Universal Robots URScript: faichun_9jan_1t1.script

def faichun_9jan_1t1():
  set_tool_communication(True, 1000000, 2, 1, 1.5, 3.5)
  set_tool_output_mode(0)
  set_tool_digital_output_mode(0, 1)
  set_tool_digital_output_mode(1, 1)
  set_tool_voltage(24)
  step_count_e741a7f4_0b30_46a8_b996_4636aff9ce90 = 0.0
  thread Step_Counter_Thread_bd4b55fe_d110_495a_a627_b98bcdc962aa():
    while (True):
      step_count_e741a7f4_0b30_46a8_b996_4636aff9ce90 = step_count_e741a7f4_0b30_46a8_b996_4636aff9ce90 + 1.0
      sync()
    end
  end
  run Step_Counter_Thread_bd4b55fe_d110_495a_a627_b98bcdc962aa()
  set_gravity([0.0, 0.0, 9.82])
  set_tcp(p[0.0,0.0,0.0,0.0,0.0,0.0])
  set_standard_analog_input_domain(0, 1)
  set_standard_analog_input_domain(1, 1)
  set_tool_analog_input_domain(0, 1)
  set_tool_analog_input_domain(1, 1)
  set_analog_outputdomain(0, 0)
  set_analog_outputdomain(1, 0)
  set_input_actions_to_default()
  set_safety_mode_transition_hardness(1)
  set_target_payload(1.070000, [0.002000, 0.003000, 0.057000], [0.001723, 0.001723, 0.001723, 0.000000, 0.000000, 0.000000])
  global B1empty=False
  global A2Empty=0
  global A1Empty=0
  global B2Empty=False
  global pallet_step=0
  global bright_box=0
  global Pallet_1_cnt=2
  global dark_boxes=0
  global Point_1=p[0.6913645118948067,-0.12399382748223003,0.49223711947071,-1.2983729986843258,1.1259514972191385,-1.2203503861141718]
  # begin: URCap Installation Node
  #   Source: External Control, 1.0.5, FZI Research Center for Information Technology
  #   Type: External Control
  # end: URCap Installation Node
  # begin: URCap Installation Node
  #   Source: OnRobot, 6.2.0, OnRobot A/S
  #   Type: OnRobot Setup
  sleep(1)
  if (False):
  end
  ON_CONN_SHIFT_BOOL = 64
  ON_CONN_SHIFT_INT = 24
  ON_CONN_SHIFT_FLOAT = 24
  ON_CONN_REG_SUM_BOOL = 0
  ON_CONN_REG_SUM_INT = 1
  ON_CONN_REG_SUM_FLOAT = 0
  ON_TOOL_SHIFT_BOOL = 64
  ON_TOOL_SHIFT_INT = 25
  ON_TOOL_SHIFT_FLOAT = 24
  ON_TOOL_SHIFT_BOOL_ARR = [64, 64, 64]
  ON_TOOL_SHIFT_INT_ARR = [25, 25, 25]
  ON_TOOL_SHIFT_FLOAT_ARR = [24, 24, 24]
  ON_TOOL_REG_SUM_BOOL = 0
  ON_TOOL_REG_SUM_INT = 0
  ON_TOOL_REG_SUM_FLOAT = 0
  ON_REGISTERS_SPEEDL_FLOAT = 0
  ON_REG_USE_TOOL = False
  ON_DI_SINGLE = 0
  ON_DI_PRIMARY = 1
  ON_DI_SECONDARY = 2
  ON_DI_DUAL = 3
  on_robot_type = 10
  on_robot_cycle = 2.0
  on_conn_ip = "localhost"
  on_tool_ip = "localhost"
  on_device_socket_port = 51234
  on_conn_xmlrpc = rpc_factory("xmlrpc", "http://localhost:41414")
  on_tool_xmlrpc = rpc_factory("xmlrpc", "http://localhost:41414")
  on_RPC = rpc_factory("xmlrpc", "http://127.0.0.1:31416")
  ON_DEBUG_LOG = False
  on_isMetric = True
  on_toolConnector = True
  on_ioqc = False
  on_dual = False
  on_computebox = False
  on_devices = 0
  on_gripper = [False, False, False]
  on_custom_tcp_id = "none"
  on_custom_tcp_enabled = False
  speedlTime = 0.001
  on_ft = False
  #======    OnRobot Globals    ======#

  ON_MATH_PI=3.141593
  ON_ZEROPOSE=p[0.0,0.0,0.0,0.0,0.0,0.0]
  ON_ZEROFRAME=p[0.0,0.0,0.0,0.0,0.0,0.0]
  ON_ZERO3D=[0.0,0.0,0.0]
  ON_ZERO6D=[0.0,0.0,0.0,0.0,0.0,0.0]
  ON_ZERO8D=[0.0,0.0,0.0,0.0,0.0,0.0,0.0,0.0]
  ON_FALSE3D=[False,False,False]
  ON_FALSE6D=[False,False,False,False,False,False]
  ON_FALSE8D=[False,False,False,False,False,False,False,False]
  global on_return=0
  on_speedL=ON_ZERO6D
  on_speedBase=ON_ZERO6D
  on_speedVect=ON_ZERO6D
  on_speedExtra=ON_ZERO6D
  on_speedCB=ON_ZERO6D
  on_speedGecko=ON_ZERO6D
  on_RTDE_error=0
  on_RTDE_tool_error=0
  on_dataProcess_thrd=0
  ON_DEVICE_ID_MISSING=0
  ON_INIT_WATCHDOG_HZ=5
  ON_INIT_TIMEOUT=2000
  on_robot_TCP_offset=ON_ZEROFRAME
  on_tcp_offset_actual=ON_ZEROFRAME
  on_cog_actual=ON_ZEROFRAME
  on_mass_actual=0.0
  on_robot_mount=[0.0,0.0]

  #======    End of OnRobot Globals    ======#
  #======    OnRobot Interface Messages    ======#

  on_devices_primary_log="OnRobot Devices"
  on_devices_secondary_log="OnRobot Secondary Device"
  on_program_halted="<br>Program halted."
  on_device_error_title="OnRobot - Device error"
  on_install_error="OnRobot Setup is not correct.<br>Check the status in the OnRobot Setup page in the Installation Tab.<br>Program halted."
  on_device_missing="No device connected.<br>Program halted."
  cb_device_missing="No OnRobot Compute Box connected.<br>Program halted."
  ft_device_missing="No OnRobot FT sensor or license detected.<br>Program halted."
  hex_device_missing="No HEX sensor connected.<br>Program halted."
  rg2ft_device_missing="No RG2-FT gripper connected.<br>Program halted."
  rg_device_missing="No RG gripper connected.<br>Program halted."
  vg_device_missing="No VG gripper connected.<br>Program halted."
  gg_device_missing="No Gecko Gripper connected.<br>Program halted."
  sg_device_missing="No Soft Gripper connected.<br>Program halted."
  tfg_device_missing="No 3FG gripper connected.<br>Program halted."
  sdr_device_missing="No OnRobot Sander connected.<br>Program halted."
  twofg_device_missing="No 2FG gripper connected.<br>Program halted."
  vgp_device_missing="No VGP gripper connected.<br>Program halted."
  mg_device_missing="No Magnetic Gripper connected.<br>Program halted."
  fgp_device_missing="No 2FGP20 Gripper connected.<br>Program halted."
  eyes_device_missing="No OnRobot Eyes connected.<br>Program halted."
  on_xmlrpc_start_ip="Connecting to OnRobot XML-RPC Server:"
  on_java_comm_error_textmsg_title="OnRobot - Communication error:"
  on_java_comm_controlsocket_open_error="Socket 'javaSocket' opening was unsuccessful."
  on_java_comm_error_title="OnRobot - Communication error"
  on_java_comm_socket_open_error="Establishing connection with the URCap was timed out.<br>Check the status in the OnRobot Setup page in the Installation Tab.<br>Program halted."
  on_rtde_feed_error_textmsg_title="OnRobot - RTDE error:"
  on_rtde_feed_error="RTDE feed error. OnRobot device count mismatch.<br>Program halted."
  on_rtde_feed_tool_error="Tool RTDE feed error. OnRobot device count mismatch.<br>Program halted."
  on_rtde_feed_open_error_textmsg="Socket 'rtdeFeed' opening was unsuccessful."
  on_rtde_feed_error_title="OnRobot - RTDE error"
  on_rtde_feed_count_error="Invalid RTDE offset setup detected. Please check RTDE Offsets at the OnRobot Setup page in the Installation Tab.<br>Program halted."
  on_rtde_feed_open_error="Establishing connection with the devices was timed out.<br>Ensure that the OnRobot devices are operational, and check the status in the OnRobot Setup page in the Installation Tab."

  #======    End of OnRobot Interface Messages    ======#
  #======    OnRobot Interface    ======#

  on_portopened_javaSocket=False
  on_rtde_feed_opened=False
  on_dataProcess_running=False
  def on_missing():
  popup(on_device_missing,title=on_device_error_title,error=True,blocking=False)
  halt
  end
  def cb_missing():
  popup(cb_device_missing,title=on_device_error_title,error=True,blocking=False)
  halt
  end
  def ft_missing():
  popup(ft_device_missing,title=on_device_error_title,error=True,blocking=False)
  halt
  end
  def hex_missing():
  popup(hex_device_missing,title=on_device_error_title,error=True,blocking=False)
  halt
  end
  def rg2ft_missing():
  popup(rg2ft_device_missing,title=on_device_error_title,error=True,blocking=False)
  halt
  end
  def rg_missing():
  popup(rg_device_missing,title=on_device_error_title,error=True,blocking=False)
  halt
  end
  def vg_missing():
  popup(vg_device_missing,title=on_device_error_title,error=True,blocking=False)
  halt
  end
  def gg_missing():
  popup(gg_device_missing,title=on_device_error_title,error=True,blocking=False)
  halt
  end
  def sg_missing():
  popup(sg_device_missing,title=on_device_error_title,error=True,blocking=False)
  halt
  end
  def tfg_missing():
  popup(tfg_device_missing,title=on_device_error_title,error=True,blocking=False)
  halt
  end
  def sdr_missing():
  popup(sdr_device_missing,title=on_device_error_title,error=True,blocking=False)
  halt
  end
  def twofg_missing():
  popup(twofg_device_missing,title=on_device_error_title,error=True,blocking=False)
  halt
  end
  def vgp_missing():
  popup(vgp_device_missing,title=on_device_error_title,error=True,blocking=False)
  halt
  end
  def mg_missing():
  popup(mg_device_missing,title=on_device_error_title,error=True,blocking=False)
  halt
  end
  def fgp_missing():
  popup(fgp_device_missing,title=on_device_error_title,error=True,blocking=False)
  halt
  end
  def eyes_missing():
  popup(eyes_device_missing,title=on_device_error_title,error=True,blocking=False)
  halt
  end
  def on_portclose_javaSocket():
  socket_close("javaSocket")
  on_portopened_javaSocket=False
  end
  def on_portopen_javaSocket():
  on_portclose_javaSocket()
  on_portopened_javaSocket=socket_open("127.0.0.1",44005,"javaSocket")
  if not on_portopened_javaSocket:
  textmsg(on_java_comm_error_textmsg_title,on_java_comm_controlsocket_open_error)
  popup(on_java_comm_socket_open_error,title=on_java_comm_error_title,error=True,blocking=False)
  halt
  end
  end
  on_conn_rtde_feed_name="rtdeFeedConn"
  on_tool_rtde_feed_name="rtdeFeedTool"
  def on_rtde_feed_close(rtdeFeedName):
  socket_close(rtdeFeedName)
  on_rtde_feed_opened=False
  end
  def on_rtde_feed_open(deviceIP,rtdeFeedName,regStart,regSum,regSpeedl):
  on_rtde_feed_close(rtdeFeedName)
  if((regStart[0]+regSum[0])>128)or((regStart[1]+regSum[1])>48)or((regStart[2]+regSum[2])>48):
  popup(on_rtde_feed_count_error,title=on_rtde_feed_error_title,error=True,blocking=False)
  textmsg(str_cat("RegStart: ",regStart),str_cat("  -  RegSum: ",regSum))
  halt
  end
  on_rtde_feed_opened=socket_open(deviceIP,on_device_socket_port,rtdeFeedName)
  if not on_rtde_feed_opened:
  on_rtde_feed_opened=socket_open(deviceIP,on_device_socket_port,rtdeFeedName)
  end
  if not on_rtde_feed_opened:
  textmsg(on_rtde_feed_error_textmsg_title,on_rtde_feed_open_error_textmsg)
  popup(on_rtde_feed_open_error,title=on_rtde_feed_error_title,error=True,blocking=False)
  halt
  end
  socket_send_int(regStart[0],rtdeFeedName)
  socket_send_int(regSum[0],rtdeFeedName)
  socket_send_int(regStart[1],rtdeFeedName)
  socket_send_int(regSum[1],rtdeFeedName)
  socket_send_int(regStart[2],rtdeFeedName)
  socket_send_int(regSum[2],rtdeFeedName)
  socket_send_int(regSpeedl,rtdeFeedName)
  socket_send_int(on_devices,rtdeFeedName)
  end
  def on_dataRead():
  enter_critical
  on_RTDE_error=read_input_integer_register(ON_CONN_SHIFT_INT)
  if(ON_REG_USE_TOOL):
  on_RTDE_tool_error=read_input_integer_register(ON_TOOL_SHIFT_INT_ARR[0])
  end
  exit_critical
  end
  def on_set_rtde_watchdog(updateHz=ON_INIT_WATCHDOG_HZ):
  local effect="stop"
  if(updateHz<1):
  effect="ignore"
  end
  watchdog_conn_reg_str=str_cat("input_int_register_",ON_CONN_SHIFT_INT)
  rtde_set_watchdog(watchdog_conn_reg_str,updateHz,effect)
  if(ON_REG_USE_TOOL):
  watchdog_tool_reg_str=str_cat("input_int_register_",ON_TOOL_SHIFT_INT_ARR[0])
  rtde_set_watchdog(watchdog_tool_reg_str,updateHz,effect)
  end
  if ON_DEBUG_LOG:
  local update_str=str_cat(" "+effect+" watchdog set to [Hz]: ",updateHz)
  textmsg(watchdog_conn_reg_str,update_str)
  if(ON_REG_USE_TOOL):
  local update_str=str_cat(" "+effect+" watchdog set to [Hz]: ",updateHz)
  textmsg(watchdog_tool_reg_str,update_str)
  end
  end
  end
  def on_speedCB_get():
  return[on_speedCB[0],on_speedCB[1],on_speedCB[2],on_speedCB[3],on_speedCB[4],on_speedCB[5]]
  end
  def on_speedGecko_get():
  local speedExtra=ON_ZERO6D
  if on_speedl_for_gecko:
  speedExtra=[on_speedGecko[0],on_speedGecko[1],on_speedGecko[2],on_speedGecko[3],on_speedGecko[4],on_speedGecko[5]]
  end
  return speedExtra
  end
  def on_speedGecko_set(speedGecko):
  on_speedGecko=[speedGecko[0],speedGecko[1],speedGecko[2],speedGecko[3],speedGecko[4],speedGecko[5]]
  end
  thread on_dataProcess_thread():
  if ON_DEBUG_LOG:
  textmsg("Starting on_dataRead thread")
  end
  local error=False
  on_dataProcess_running=True
  sync()
  while on_dataProcess_running:
  sync()
  on_dataRead()
  error=on_error((on_RTDE_error<0),on_rtde_feed_error,on_rtde_feed_error_title,error)
  error=on_error((ON_REG_USE_TOOL and(on_RTDE_tool_error<0)),on_rtde_feed_tool_error,on_rtde_feed_error_title,error)
  on_dataProcess_running=not error
  end
  if error:
  halt
  end
  if ON_DEBUG_LOG:
  textmsg("Stopping on_dataRead thread")
  end
  end
  thread on_set_watchdog_thread():
  sleep(2)
  on_set_rtde_watchdog(updateHz=ON_INIT_WATCHDOG_HZ)
  sleep(1/ON_INIT_WATCHDOG_HZ)
  on_dataProcess_running=False
  kill on_dataProcess_thrd
  end

  #======    End of OnRobot Interface    ======#
  #======    OnRobot QC Setup Tool Connector    ======#

  def tc_setup_tool():
  if ON_DEBUG_LOG:
  textmsg("QC Setup Tool Connector start...")
  end
  set_tool_voltage(24)

  set_tool_communication(True,1000000,2,1,1.5,3.5)

  if ON_DEBUG_LOG:
  textmsg("QC Setup Tool Connector end.")
  end
  end

  #======    End of OnRobot QC Setup Tool Connector    ======#
  #======    OnRobot TCP Messages    ======#

  on_tcp_log_msg_default="OnRobot: Robot TCP Offset set to:"
  on_tcp_log_msg_primary="OnRobot: Robot TCP Offset set to Primary:"
  on_tcp_log_msg_secondary="OnRobot: Robot TCP Offset set to Secondary:"

  #======    End of OnRobot TCP Messages    ======#
  #======    OnRobot TCP    ======#

  on_tcp_offset_actual=ON_ZEROFRAME
  on_tcp_offset_primary=ON_ZEROFRAME
  on_tcp_static_primary=ON_ZEROFRAME
  on_tcp_dynamic_primary=ON_ZEROFRAME
  on_tcp_adapters=ON_ZEROFRAME
  on_tcp_qc_primary=ON_ZEROFRAME
  on_tcp_base_primary=ON_ZEROFRAME
  on_tcp_gripper_static_primary=ON_ZEROFRAME
  on_tcp_workpiece_primary=ON_ZEROFRAME
  on_tcp_gripper_dynamic_primary=ON_ZEROFRAME
  on_tcp_gripper_primary=ON_ZEROFRAME
  on_tcp_offset_secondary=ON_ZEROFRAME
  on_tcp_static_secondary=ON_ZEROFRAME
  on_tcp_dynamic_secondary=ON_ZEROFRAME
  on_tcp_qc_secondary=ON_ZEROFRAME
  on_tcp_base_secondary=ON_ZEROFRAME
  on_tcp_gripper_static_secondary=ON_ZEROFRAME
  on_tcp_workpiece_secondary=ON_ZEROFRAME
  on_tcp_gripper_dynamic_secondary=ON_ZEROFRAME
  on_tcp_gripper_secondary=ON_ZEROFRAME
  on_tcp_custom_preset_assigned=False
  on_tcp_custom_preset=ON_ZEROFRAME
  def on_tcp_init_adapters():
  if ON_DEBUG_LOG:
  textmsg("TCP Init Adapters start..")
  end
  enter_critical
  on_tcp_adapters=ON_ZEROFRAME
  local adapterCount=length(on_tcp_adapters_array)
  local i=0
  while(i<adapterCount):
  on_tcp_adapters=pose_trans(on_tcp_adapters,on_tcp_adapters_array[i])
  i=i+1
  end
  exit_critical
  if ON_DEBUG_LOG:
  textmsg("TCP Init Adapters end.")
  end
  end
  def on_tcp_update_primary():
  if ON_DEBUG_LOG:
  textmsg("TCP Update Primary start..")
  end
  on_tcp_gripper_dynamic_primary=p[0.0, 0.0, 0.0, 0.0, 0.0, 0.0]
  enter_critical
  on_tcp_dynamic_primary=pose_trans(on_tcp_static_primary,on_tcp_gripper_dynamic_primary)
  on_tcp_offset_primary=pose_trans(on_tcp_dynamic_primary,on_tcp_workpiece_primary)
  exit_critical
  if ON_DEBUG_LOG:
  textmsg("TCP Update Primary end.")
  end
  end
  def on_tcp_init_primary():
  if ON_DEBUG_LOG:
  textmsg("TCP Init Primary start..")
  end
  enter_critical
  on_tcp_base_primary=pose_trans(on_tcp_adapters,on_tcp_qc_primary)
  on_tcp_static_primary=pose_trans(on_tcp_base_primary,on_tcp_gripper_static_primary)
  exit_critical
  on_tcp_update_primary()
  if ON_DEBUG_LOG:
  textmsg("TCP Init Primary end.")
  end
  end
  def on_tcp_offset_set(TCP_offset):
  if ON_DEBUG_LOG:
  textmsg("TCP Offset set started!")
  end
  on_tcp_offset_send(TCP_offset)
  if(on_follow_tcp):
  set_tcp(TCP_offset)
  end
  on_robot_TCP_offset=TCP_offset
  if ON_DEBUG_LOG:
  textmsg("TCP Offset set to: ",on_robot_TCP_offset)
  end
  end
  def on_tcp_offset_forced_set_actual(isPrimary=True):
  if(not on_follow_tcp):

  local tcp_log_msg=on_tcp_log_msg_default

  textmsg(tcp_log_msg,on_tcp_offset_actual)
  set_tcp(on_tcp_offset_actual)
  end
  end
  def on_tcp_update(isPrimary=True):
  on_tcp_update_primary()

  on_tcp_set_actual_to(isPrimary)
  end
  def on_tcp_set_actual_to(isPrimary=True):

  on_tcp_offset_actual=on_tcp_offset_primary
  if(on_follow_tcp):
  textmsg(on_tcp_log_msg_default,on_tcp_offset_actual)
  end

  on_tcp_active_is_primary=isPrimary
  on_tcp_offset_set(on_tcp_offset_actual)
  end
  def on_tcp_update_workpiece_primary(workpiece_offset):
  if ON_DEBUG_LOG:
  textmsg("TCP Update Tool Primary start..")
  end
  on_tcp_workpiece_primary=workpiece_offset
  on_tcp_update_primary()
  if ON_DEBUG_LOG:
  textmsg("TCP Update Tool Primary end.")
  end
  end
  def on_tcp_workpiece_rpy_get(xyz=[0.0,0.0,0.0],rpy=[0.0,0.0,0.0]):
  local rotvec=rpy2rotvec(rpy)
  local workpiece_offset=p[xyz[0],xyz[1],xyz[2],rotvec[0],rotvec[1],rotvec[2]]
  return workpiece_offset
  end

  def on_tcp_update_workpiece(workpiece_offset,tool_index=0):
  if ON_DEBUG_LOG:
  textmsg("TCP Update Tool start..")
  end
  if(tool_index!=ON_DI_SECONDARY):
  on_tcp_update_workpiece_primary(workpiece_offset)
  local isPrimary=True

  end
  on_tcp_set_actual_to(isPrimary)
  if ON_DEBUG_LOG:
  textmsg("TCP Update Tool end.")
  end
  end
  def on_get_tcp_for(tool_index):
  if tool_index==ON_DI_SECONDARY:
  local actual_tcp=on_tcp_static_secondary
  else:
  local actual_tcp=on_tcp_static_primary
  end
  return actual_tcp
  end
  def on_tcp_custom_unused():
  return ON_ZEROFRAME
  end
  def on_tcp_update_custom():
  if ON_DEBUG_LOG:
  textmsg("TCP Update Custom start..")
  end
  if(on_custom_tcp_enabled):
  on_tcp_custom_unused()
  on_tcp_custom_unused()
  on_tcp_custom_unused()
  on_tcp_custom_unused()

  end
  if ON_DEBUG_LOG:
  textmsg("TCP Update Custom end.")
  end
  end

  #======    End of OnRobot TCP    ======#
  #======    OnRobot Payload Messages    ======#

  on_mass_log_msg="OnRobot: Robot Payload Mass set to:"
  on_cog_log_msg="OnRobot: Robot Payload Center of Gravity set to:"

  #======    End of OnRobot Payload Messages    ======#
  #======    OnRobot Payload    ======#

  on_cog_actual=ON_ZEROFRAME
  on_mass_actual=0.0
  on_cog_primary=ON_ZEROFRAME
  on_cog_L1L2_primary=ON_ZEROFRAME
  on_mass_primary=0.0
  on_mass_L1L2_primary=0.0
  on_cog_adapters=ON_ZEROFRAME
  on_cog_qc_primary=ON_ZEROFRAME
  on_cog_base_primary=ON_ZEROFRAME
  on_cog_gripper_primary=ON_ZEROFRAME
  on_cog_workpiece_primary=ON_ZEROFRAME
  on_mass_adapters=0.0
  on_mass_qc_primary=0.0
  on_mass_base_primary=0.0
  on_mass_gripper_primary=0.0
  on_mass_workpiece_primary=0.0
  on_cog_secondary=ON_ZEROFRAME
  on_mass_secondary=0.0
  on_cog_gripper_secondary=ON_ZEROFRAME
  on_mass_gripper_secondary=0.0
  on_cog_workpiece_secondary=ON_ZEROFRAME
  on_mass_workpiece_secondary=0.0
  ON_LB2KG001=0.45359237/100
  def on_payload_init_adapters():
  if ON_DEBUG_LOG:
  textmsg("TCP Init Adapters start..")
  end
  enter_critical
  on_cog_adapters=ON_ZEROFRAME
  on_mass_adapters=0.0
  local massLAL0Ratio=0
  local adapterAbsCOG=ON_ZEROFRAME
  local tcp_adapter_offset=ON_ZEROFRAME
  local adapterCount=length(on_tcp_adapters_array)
  local i=0
  while(i<adapterCount):
  on_mass_adapters=on_mass_adapters+on_mass_adapters_array[i]
  if(on_mass_adapters<=0):
  massLAL0Ratio=0
  else:
  massLAL0Ratio=on_mass_adapters_array[i]/on_mass_adapters
  end
  adapterAbsCOG=pose_trans(tcp_adapter_offset,on_tcp_adapters_array[i])
  adapterAbsCOG=p[adapterAbsCOG[0],adapterAbsCOG[1],adapterAbsCOG[2],0.0,0.0,0.0]
  on_cog_adapters=interpolate_pose(on_cog_adapters,adapterAbsCOG,massLAL0Ratio)
  on_cog_adapters=p[on_cog_adapters[0],on_cog_adapters[1],on_cog_adapters[2],0.0,0.0,0.0]
  tcp_adapter_offset=pose_trans(tcp_adapter_offset,on_tcp_adapters_array[i])
  i=i+1
  sync()
  end
  exit_critical
  if ON_DEBUG_LOG:
  textmsg("TCP Init Adapters end.")
  end
  end
  def on_payload_update_primary():
  if ON_DEBUG_LOG:
  textmsg("Payload Update Primary start..")
  end
  enter_critical
  on_mass_primary=on_mass_L1L2_primary+on_mass_workpiece_primary
  local massL1L2L3Ratio=on_mass_workpiece_primary/on_mass_primary
  local workpieceAbsCOG=pose_trans(on_tcp_dynamic_primary,on_cog_workpiece_primary)
  workpieceAbsCOG=p[workpieceAbsCOG[0],workpieceAbsCOG[1],workpieceAbsCOG[2],0.0,0.0,0.0]
  on_cog_primary=interpolate_pose(on_cog_L1L2_primary,workpieceAbsCOG,massL1L2L3Ratio)
  on_cog_primary=p[on_cog_primary[0],on_cog_primary[1],on_cog_primary[2],0.0,0.0,0.0]
  exit_critical
  if ON_DEBUG_LOG:
  textmsg("Payload Update Primary end.")
  end
  end
  def on_payload_init_primary():
  if ON_DEBUG_LOG:
  textmsg("Payload Init Primary start..")
  end
  enter_critical
  on_mass_base_primary=on_mass_adapters+on_mass_qc_primary
  local massL0L1Ratio=on_mass_qc_primary/on_mass_base_primary
  on_mass_L1L2_primary=on_mass_base_primary+on_mass_gripper_primary
  local massL1L2Ratio=on_mass_gripper_primary/on_mass_L1L2_primary
  local qcAbsCOG=pose_trans(on_tcp_adapters,on_cog_qc_primary)
  qcAbsCOG=p[qcAbsCOG[0],qcAbsCOG[1],qcAbsCOG[2],0.0,0.0,0.0]
  on_cog_base_primary=interpolate_pose(on_cog_adapters,qcAbsCOG,massL0L1Ratio)
  on_cog_base_primary=p[on_cog_base_primary[0],on_cog_base_primary[1],on_cog_base_primary[2],0.0,0.0,0.0]
  local gripperAbsCOG=pose_trans(on_tcp_base_primary,on_cog_gripper_primary)
  gripperAbsCOG=p[gripperAbsCOG[0],gripperAbsCOG[1],gripperAbsCOG[2],0.0,0.0,0.0]
  on_cog_L1L2_primary=interpolate_pose(on_cog_base_primary,gripperAbsCOG,massL1L2Ratio)
  on_cog_L1L2_primary=p[on_cog_L1L2_primary[0],on_cog_L1L2_primary[1],on_cog_L1L2_primary[2],0.0,0.0,0.0]
  exit_critical
  on_payload_update_primary()
  if ON_DEBUG_LOG:
  textmsg("Payload Init Primary end.")
  end
  end
  def on_payload_update():
  on_payload_update_primary()

  on_mass_actual =on_mass_primary
  on_cog_actual=on_cog_primary

  on_payload_set_actual()
  end
  def on_payload_set_actual():

  on_mass_actual =on_mass_primary
  on_cog_actual=on_cog_primary

  local CoG=[on_cog_actual[0],on_cog_actual[1],on_cog_actual[2]]
  on_payload_set(on_mass_actual,CoG)
  end
  def on_payload_update_workpiece_primary(workpiece_mass=0,workpiece_cog=[0.0,0.0,0.0]):
  if ON_DEBUG_LOG:
  textmsg("Payload Update Workpiece Primary start..")
  end
  on_cog_workpiece_primary=p[workpiece_cog[0],workpiece_cog[1],workpiece_cog[2],0.0,0.0,0.0]
  on_mass_workpiece_primary=workpiece_mass
  on_payload_update_primary()
  if ON_DEBUG_LOG:
  textmsg("Payload Update Workpiece Primary end.")
  end
  end
  def on_payload_set(mass,CoG):
  if ON_DEBUG_LOG:
  textmsg("Payload set started!")
  end
  local center_of_gravity=[CoG[0],CoG[1],CoG[2]]
  on_payload_send(center_of_gravity,mass)
  if(on_isMetric):
  local roundedMass=floor(mass*100+0.5)/100
  else:
  local roundedMass=floor(mass/ON_LB2KG001+0.5)*ON_LB2KG001
  end
  set_payload(roundedMass,center_of_gravity)
  on_mass_actual=roundedMass
  on_cog_actual=p[CoG[0],CoG[1],CoG[2],0.0,0.0,0.0]
  if ON_DEBUG_LOG:
  textmsg("Payload mass, CoG set to: ",str_cat(str_cat(mass,", "),CoG))
  end
  end

  def on_payload_update_secondary():
  end
  def on_payload_init_secondary():
  end

  def on_payload_update_workpiece(workpiece_mass,workpiece_cog=[0.0,0.0,0.0],tool_index=0):
  if ON_DEBUG_LOG:
  textmsg("Payload Update Workpiece start..")
  end
  if(tool_index!=ON_DI_SECONDARY):
  on_cog_workpiece_primary=p[workpiece_cog[0],workpiece_cog[1],workpiece_cog[2],0.0,0.0,0.0]
  on_mass_workpiece_primary=workpiece_mass
  else:
  on_cog_workpiece_secondary=p[workpiece_cog[0],workpiece_cog[1],workpiece_cog[2],0.0,0.0,0.0]
  on_mass_workpiece_secondary=workpiece_mass
  end
  on_payload_update()
  if ON_DEBUG_LOG:
  textmsg("Payload Update Workpiece end.")
  end
  end
  def on_payload_get_cog2tcp_workpiece(tool_index=0):
  if(tool_index!=ON_DI_SECONDARY):
  local cog_tool=[on_tcp_workpiece_primary[0],on_tcp_workpiece_primary[1],on_tcp_workpiece_primary[2]]
  else:
  local cog_tool=[on_tcp_workpiece_secondary[0],on_tcp_workpiece_secondary[1],on_tcp_workpiece_secondary[2]]
  end
  return cog_tool
  end

  #======    End of OnRobot Payload    ======#
  #======    OnRobot QC TCP    ======#

  onrobotmini=0

  def on_tcp_offset_send(TCP_offset):
  on_robot_TCP_offset=TCP_offset
  end
  def on_payload_send(CoG,mass):
  on_robot_payload_cog=CoG
  on_robot_payload_mass=mass
  end


  #======    End of OnRobot QC TCP    ======#
  #======    OnRobot  Speedl    ======#

  on_speedl_thread_handler=0
  on_speedl_is_enabled=False
  on_speedl_is_running=False
  on_speedl_acc=0.0
  ft_speedl_hg_caranteen_reached=False
  ft_speedl_hg_caranteen_safemode=False
  on_speedl_for_ftcontrol=False
  on_speedl_for_move=False
  on_speedl_for_handguide=False
  on_speedl_for_insertpart=False
  on_speedl_for_depthcompensation=False
  on_speedl_for_center=False
  on_speedl_for_gecko=False
  on_speedl_acc=10000.0
  on_speedl_acc_to_zero=3.0
  ON_SPEEDL_FTCONTROL=1
  ON_SPEEDL_HANDGUIDE=2
  ON_SPEEDL_TRAJECTORY=3
  ON_SPEEDL_MOVE=ON_SPEEDL_TRAJECTORY
  ON_SPEEDL_INSERTPART=4
  ON_SPEEDL_DEPTHCOMP=5
  ON_SPEEDL_CENTER=6
  ON_SPEEDL_GECKO=7
  def on_wait_ms(time_ms):
  local sync_time=ceil(norm(time_ms/2.0))
  while(sync_time>0):
  sync_time=sync_time-1
  sync()
  end
  end
  def on_error(status_flag,message,title,stop_var=False):
  if(status_flag):
  popup(message,title=title,error=True,blocking=False)
  stop_var=True
  end
  return stop_var
  end
  def on_warning(status_flag,message,title,isPopupNeeded=False,is_shown=False):
  if(status_flag):
  if(not is_shown):
  if(isPopupNeeded):
  popup(message,title=title,warning=True,blocking=False)
  else:
  textmsg(title+": ",message)
  end
  is_shown=True
  end
  else:
  is_shown=False
  end
  return is_shown
  end
  def on_speedl_add_extra(speedBase,speedExtra):
  speedSum=ON_ZERO6D
  speedBaseP=p[speedBase[0],speedBase[1],speedBase[2],speedBase[3],speedBase[4],speedBase[5]]
  speedExtraP=p[speedExtra[0],speedExtra[1],speedExtra[2],speedExtra[3],speedExtra[4],speedExtra[5]]
  speedSumP=pose_add(speedExtraP,speedBaseP)
  speedSum=[speedSumP[0],speedSumP[1],speedSumP[2],speedSumP[3],speedSumP[4],speedSumP[5]]
  return speedSum
  end

  thread on_speedl_thread():
  if ON_DEBUG_LOG:
  textmsg("Speedl thread started..")
  end
  enter_critical
  on_speedl_is_running=True
  on_speedl_is_enabled=True
  exit_critical
  on_speedL=ON_ZERO6D
  on_speedL_last=ON_ZERO6D

  while on_speedl_is_running:
  on_speedBase=on_speedCB_get()
  on_speedL=on_speedBase


  if on_speedl_is_enabled:
  if(on_speedL==ON_ZERO6D):
  on_speedL=[on_speedL_last[0]/100,on_speedL_last[1]/100,on_speedL_last[2]/100,on_speedL_last[3]/100,on_speedL_last[4]/100,on_speedL_last[5]/100]
  end
  speedl(on_speedL,a=on_speedl_acc,t=speedlTime)
  else:
  speedl(ON_ZERO6D,a=on_speedl_acc_to_zero,t=speedlTime)
  end
  on_speedL_last=on_speedL
  end

  on_speedL=ON_ZERO6D
  if ON_DEBUG_LOG:
  textmsg("Speedl thread ended.")
  end
  end
  def on_speedl_integer_get():
  local speedl_integer=binary_list_to_integer([on_speedl_for_ftcontrol,on_speedl_for_handguide,on_speedl_for_move,on_speedl_for_insertpart,on_speedl_for_depthcompensation,on_speedl_for_center,on_speedl_for_gecko])
  return speedl_integer
  end
  def on_speedl_start_for(speedl_id):
  if(speedl_id==ON_SPEEDL_FTCONTROL):
  on_speedl_for_ftcontrol=True
  elif(speedl_id==ON_SPEEDL_HANDGUIDE):
  on_speedl_for_handguide=True
  elif(speedl_id==ON_SPEEDL_TRAJECTORY):
  on_speedl_for_move=True
  elif(speedl_id==ON_SPEEDL_INSERTPART):
  on_speedl_for_insertpart=True
  elif(speedl_id==ON_SPEEDL_DEPTHCOMP):
  on_speedl_for_depthcompensation=True
  elif(speedl_id==ON_SPEEDL_CENTER):
  on_speedl_for_center=True
  elif(speedl_id==ON_SPEEDL_GECKO):
  on_speedl_for_gecko=True
  else:
  textmsg("Unknown Start speedl ID received: ",speedl_id)
  end
  local speedl_integer=on_speedl_integer_get()
  if not(speedl_integer==0):
  if not on_speedl_is_running:
  on_speedl_thread_handler=run on_speedl_thread()
  end
  end
  return on_speedl_is_running
  end
  def on_speedl_stop_for(speedl_id,brake=10,brakeRot=10):
  if(speedl_id==ON_SPEEDL_FTCONTROL):
  on_speedl_for_ftcontrol=False
  elif(speedl_id==ON_SPEEDL_HANDGUIDE):
  on_speedl_for_handguide=False
  elif(speedl_id==ON_SPEEDL_TRAJECTORY):
  on_speedl_for_move=False
  elif(speedl_id==ON_SPEEDL_INSERTPART):
  on_speedl_for_insertpart=False
  elif(speedl_id==ON_SPEEDL_DEPTHCOMP):
  on_speedl_for_depthcompensation=False
  elif(speedl_id==ON_SPEEDL_CENTER):
  on_speedl_for_center=False
  elif(speedl_id==ON_SPEEDL_GECKO):
  on_speedl_for_gecko=False
  on_speedGecko_set(ON_ZERO6D)
  else:
  textmsg("Unknown Stop speedl ID received: ",speedl_id)
  end
  local speedl_integer=on_speedl_integer_get()
  if(speedl_integer==0):
  if(on_speedl_is_running):
  kill on_speedl_thread_handler
  enter_critical
  on_speedl_is_running=False
  exit_critical

  end
  if ON_DEBUG_LOG:
  textmsg("Speedl thread stopped")
  end
  stopl(brake,brakeRot)
  end
  return on_speedl_is_running
  end
  def on_speedl_pause():
  on_speedl_is_enabled=False
  return on_speedl_integer_get()
  end
  def on_speedl_resume():
  on_speedl_is_enabled=True
  return on_speedl_integer_get()
  end

  #======    End of OnRobot  Speedl    ======#
  textmsg(on_devices_primary_log, ": Quick Changer + QC Tool Side + [0.0, 0.0, 0.0, 0.0, 0.0, 0.0]")
  on_follow_tcp = False
  on_tcp_active_is_primary = True
  on_tcp_adapters_array = []
  on_cog_adapters_array = []
  on_mass_adapters_array = []
  on_tcp_qc_primary = p[0.0, 0.0, 0.0136, 0.0, 0.0, 0.0]
  on_cog_qc_primary = p[0.0, 0.0, 0.004, 0.0, 0.0, 0.0]
  on_mass_qc_primary = 0.06
  on_tcp_gripper_static_primary = p[0.0, 0.0, 0.017, 0.0, 0.0, 0.0]
  on_cog_gripper_primary = p[0.0, 0.0, 0.002, 0.0, 0.0, 0.0]
  on_mass_gripper_primary = 0.14
  on_tcp_workpiece_primary = p[0.0, 0.0, 0.0, 0.0, 0.0, 0.0]
  on_cog_workpiece_primary = p[0.0, 0.0, 0.0, 0.0, 0.0, 0.0]
  on_mass_workpiece_primary = 0.0
  #======    OnRobot Run    ======#

  on_portopen_javaSocket()
  sync()
  textmsg(on_xmlrpc_start_ip,on_conn_ip)
  if(ON_REG_USE_TOOL):
  on_regStart_conn=[ON_CONN_SHIFT_BOOL,ON_CONN_SHIFT_INT,ON_CONN_SHIFT_FLOAT]
  on_regSum_conn=[ON_CONN_REG_SUM_BOOL,ON_CONN_REG_SUM_INT,ON_CONN_REG_SUM_FLOAT]
  on_rtde_feed_open(on_conn_ip,on_conn_rtde_feed_name,on_regStart_conn,on_regSum_conn,ON_REGISTERS_SPEEDL_FLOAT)
  sync()
  textmsg(on_xmlrpc_start_ip,on_tool_ip)
  on_regStart_tool=[ON_TOOL_SHIFT_BOOL,ON_TOOL_SHIFT_INT,ON_TOOL_SHIFT_FLOAT]
  on_regSum_tool=[ON_TOOL_REG_SUM_BOOL,ON_TOOL_REG_SUM_INT,ON_TOOL_REG_SUM_FLOAT]
  on_rtde_feed_open(on_tool_ip,on_tool_rtde_feed_name,on_regStart_tool,on_regSum_tool,0)
  sync()
  else:
  on_regStart_conn=[ON_CONN_SHIFT_BOOL,ON_CONN_SHIFT_INT,ON_CONN_SHIFT_FLOAT]
  on_regSum_conn=[ON_CONN_REG_SUM_BOOL,ON_CONN_REG_SUM_INT,ON_CONN_REG_SUM_FLOAT]
  on_rtde_feed_open(on_conn_ip,on_conn_rtde_feed_name,on_regStart_conn,on_regSum_conn,ON_REGISTERS_SPEEDL_FLOAT)
  sync()
  end
  on_set_rtde_watchdog(updateHz=0.2)
  sync()
  on_dataProcess_thrd=run on_dataProcess_thread()
  sync()
  on_tcp_init_adapters()
  on_payload_init_adapters()
  on_tcp_init_primary()
  on_payload_init_primary()

  on_tcp_update_custom()
  on_tcp_set_actual_to(on_tcp_active_is_primary)
  if(on_follow_tcp):
  on_payload_set_actual()
  end
  on_watchdog_thrd=run on_set_watchdog_thread()
  sync()
  def done_waiting_for_init(device_name,product_code,tool_index=0):
  textmsg(str_cat(device_name,str_cat(str_cat("[",tool_index),"]: ")),product_code)
  end

  #======    End of OnRobot Run    ======#
  #======    OnRobot QC Start    ======#

  if(on_toolConnector):
  tc_setup_tool()
  end
  sync()

  #======    End of OnRobot QC Start    ======#
  # end: URCap Installation Node
  $ 1 "Robot Program"
  $ 2 "Script: FaiChun_9 Jan_11_2_t1.script"
  def Machining1():
    # Default parameters:
    global speed_ms = 0.05
    global speed_rads = 0.75
    global accel_mss = 3
    global accel_radss = 1.2
    global blend_radius_m = 0.0003

    # Add subprograms here
    # Start of main program
    # Program generated by RoboDK v5.6.8 for UR10e on 17/01/2025 15:24:14
    # Using nominal kinematics.
    blend_radius_m = 0.0003
    speed_ms = 0.05
    # set_reference(p[0.340000, -0.240000, 0.001500, 0.000000, 0.000000, 0.000000])
    set_tcp(p[0.000000, 0.000000, 0.252000, 0.000000, 0.000000, 0.000000])
    # Show Tool
    movej([0.140721, -1.398447, -2.445688, -0.868253, 1.570796, 1.711517],accel_radss,speed_rads,0,blend_radius_m)
    movel([0.140721, -1.451124, -2.475554, -0.785711, 1.570796, 1.711517],accel_mss,speed_ms,0,blend_radius_m)
    #SetTool1
    #M_RunCode6
    #SetRPM60000
    speed_ms = 0.05
    #M_RunCode3
    movel([0.140721, -1.474076, -2.486639, -0.751674, 1.570796, 1.711517],accel_mss,speed_ms,0,blend_radius_m)
    speed_ms = 0.003
    movel([0.140721, -1.480003, -2.489338, -0.743048, 1.570796, 1.711517],accel_mss,speed_ms,0,blend_radius_m)
    speed_ms = 0.02
    movel([-0.135603, -1.563113, -2.412732, -0.736544, 1.570796, 1.435194],accel_mss,speed_ms,0,blend_radius_m)
    movel([-0.182919, -1.334068, -2.598334, -0.779987, 1.570796, 1.387878],accel_mss,speed_ms,0,blend_radius_m)
    movel([0.198662, -1.168946, -2.687374, -0.856069, 1.570796, 1.769459],accel_mss,speed_ms,0,blend_radius_m)
    movel([0.140721, -1.480003, -2.489338, -0.743048, 1.570796, 1.711517],accel_mss,speed_ms,0,blend_radius_m)
    speed_ms = 0.003
    movel([0.140721, -1.474076, -2.486639, -0.751674, 1.570796, 1.711517],accel_mss,speed_ms,0,blend_radius_m)
    speed_ms = 0.05
    movel([0.140721, -1.451124, -2.475554, -0.785711, 1.570796, 1.711517],accel_mss,speed_ms,0,blend_radius_m)
    #M_RunCode9
    movel([0.136570, -1.444454, -2.480985, -0.786951, 1.570796, 1.707367],accel_mss,speed_ms,0,blend_radius_m)
    #M_RunCode3
    movel([0.136570, -1.467543, -2.492148, -0.752698, 1.570796, 1.707367],accel_mss,speed_ms,0,blend_radius_m)
    speed_ms = 0.003
    movel([0.136570, -1.473508, -2.494867, -0.744014, 1.570796, 1.707367],accel_mss,speed_ms,0,blend_radius_m)
    speed_ms = 0.012
    movel([0.132210, -1.474416, -2.494098, -0.743875, 1.570796, 1.703007],accel_mss,speed_ms,0,blend_radius_m)
    movel([0.131633, -1.478168, -2.490906, -0.743314, 1.570796, 1.702429],accel_mss,speed_ms,0,blend_radius_m)
    movel([0.125209, -1.479526, -2.489746, -0.743117, 1.570796, 1.696006],accel_mss,speed_ms,0,blend_radius_m)
    movel([0.125756, -1.475786, -2.492935, -0.743668, 1.570796, 1.696552],accel_mss,speed_ms,0,blend_radius_m)
    movel([0.123495, -1.476273, -2.492521, -0.743595, 1.570796, 1.694292],accel_mss,speed_ms,0,blend_radius_m)
    movel([0.122957, -1.480010, -2.489332, -0.743047, 1.570796, 1.693753],accel_mss,speed_ms,0,blend_radius_m)
    movel([0.117581, -1.481181, -2.488328, -0.742880, 1.570796, 1.688377],accel_mss,speed_ms,0,blend_radius_m)
    movel([0.116539, -1.481408, -2.488133, -0.742848, 1.570796, 1.687335],accel_mss,speed_ms,0,blend_radius_m)
    movel([0.117294, -1.475890, -2.492847, -0.743652, 1.570796, 1.688091],accel_mss,speed_ms,0,blend_radius_m)
    movel([0.121657, -1.474929, -2.493663, -0.743797, 1.570796, 1.692454],accel_mss,speed_ms,0,blend_radius_m)
    movel([0.121935, -1.472979, -2.495315, -0.744096, 1.570796, 1.692731],accel_mss,speed_ms,0,blend_radius_m)
    movel([0.115294, -1.474450, -2.494069, -0.743870, 1.570796, 1.686091],accel_mss,speed_ms,0,blend_radius_m)
    movel([0.114291, -1.481907, -2.487705, -0.742777, 1.570796, 1.685087],accel_mss,speed_ms,0,blend_radius_m)
    movel([0.113249, -1.482141, -2.487504, -0.742744, 1.570796, 1.684045],accel_mss,speed_ms,0,blend_radius_m)
    speed_ms = 0.02
    movel([-0.001403, -1.512452, -2.460728, -0.739209, 1.570796, 1.569393],accel_mss,speed_ms,0,blend_radius_m)
    movel([-0.112335, -1.550651, -2.424918, -0.736820, 1.570796, 1.458461],accel_mss,speed_ms,0,blend_radius_m)
    speed_ms = 0.012
    movel([-0.113250, -1.544354, -2.430981, -0.737054, 1.570796, 1.457547],accel_mss,speed_ms,0,blend_radius_m)
    movel([-0.119333, -1.546716, -2.428713, -0.736959, 1.570796, 1.451463],accel_mss,speed_ms,0,blend_radius_m)
    movel([-0.119087, -1.548345, -2.427145, -0.736899, 1.570796, 1.451710],accel_mss,speed_ms,0,blend_radius_m)
    movel([-0.115090, -1.546793, -2.428639, -0.736956, 1.570796, 1.455706],accel_mss,speed_ms,0,blend_radius_m)
    movel([-0.114409, -1.551442, -2.424151, -0.736796, 1.570796, 1.456387],accel_mss,speed_ms,0,blend_radius_m)
    movel([-0.115366, -1.551811, -2.423794, -0.736784, 1.570796, 1.455430],accel_mss,speed_ms,0,blend_radius_m)
    movel([-0.120291, -1.553718, -2.421942, -0.736729, 1.570796, 1.450506],accel_mss,speed_ms,0,blend_radius_m)
    movel([-0.120772, -1.550599, -2.424968, -0.736822, 1.570796, 1.450025],accel_mss,speed_ms,0,blend_radius_m)
    movel([-0.122835, -1.551404, -2.424188, -0.736797, 1.570796, 1.447961],accel_mss,speed_ms,0,blend_radius_m)
    movel([-0.122346, -1.554519, -2.421162, -0.736708, 1.570796, 1.448450],accel_mss,speed_ms,0,blend_radius_m)
    movel([-0.128198, -1.556814, -2.418922, -0.736653, 1.570796, 1.442598],accel_mss,speed_ms,0,blend_radius_m)
    movel([-0.128709, -1.553718, -2.421941, -0.736729, 1.570796, 1.442088],accel_mss,speed_ms,0,blend_radius_m)
    movel([-0.132665, -1.555290, -2.420410, -0.736688, 1.570796, 1.438132],accel_mss,speed_ms,0,blend_radius_m)
    movel([-0.133450, -1.550705, -2.424865, -0.736819, 1.570796, 1.437347],accel_mss,speed_ms,0,blend_radius_m)
    movel([-0.129474, -1.549116, -2.426401, -0.736872, 1.570796, 1.441323],accel_mss,speed_ms,0,blend_radius_m)
    movel([-0.129743, -1.547498, -2.427961, -0.736930, 1.570796, 1.441053],accel_mss,speed_ms,0,blend_radius_m)
    movel([-0.133727, -1.549091, -2.426425, -0.736873, 1.570796, 1.437069],accel_mss,speed_ms,0,blend_radius_m)
    movel([-0.134396, -1.545231, -2.430140, -0.737018, 1.570796, 1.436400],accel_mss,speed_ms,0,blend_radius_m)
    movel([-0.134524, -1.544477, -2.430863, -0.737049, 1.570796, 1.436272],accel_mss,speed_ms,0,blend_radius_m)
    movel([-0.128589, -1.542092, -2.433143, -0.737154, 1.570796, 1.442208],accel_mss,speed_ms,0,blend_radius_m)
    movel([-0.128072, -1.545228, -2.430143, -0.737018, 1.570796, 1.442725],accel_mss,speed_ms,0,blend_radius_m)
    movel([-0.125992, -1.544401, -2.430936, -0.737052, 1.570796, 1.444805],accel_mss,speed_ms,0,blend_radius_m)
    movel([-0.126769, -1.539625, -2.435492, -0.737272, 1.570796, 1.444027],accel_mss,speed_ms,0,blend_radius_m)
    movel([-0.134806, -1.542853, -2.432416, -0.737120, 1.570796, 1.435990],accel_mss,speed_ms,0,blend_radius_m)
    movel([-0.151268, -1.454119, -2.510984, -0.747286, 1.570796, 1.419528],accel_mss,speed_ms,0,blend_radius_m)
    speed_ms = 0.02
    movel([-0.171874, -1.356528, -2.583560, -0.772301, 1.570796, 1.398922],accel_mss,speed_ms,0,blend_radius_m)
    movel([-0.172081, -1.355600, -2.584184, -0.772605, 1.570796, 1.398715],accel_mss,speed_ms,0,blend_radius_m)
    speed_ms = 0.012
    movel([-0.162028, -1.350393, -2.587664, -0.774332, 1.570796, 1.408769],accel_mss,speed_ms,0,blend_radius_m)
    movel([-0.163290, -1.344436, -2.591600, -0.776353, 1.570796, 1.407507],accel_mss,speed_ms,0,blend_radius_m)
    movel([-0.165922, -1.345805, -2.590700, -0.775884, 1.570796, 1.404874],accel_mss,speed_ms,0,blend_radius_m)
    movel([-0.165080, -1.349718, -2.588113, -0.774558, 1.570796, 1.405716],accel_mss,speed_ms,0,blend_radius_m)
    movel([-0.172527, -1.353588, -2.585533, -0.773268, 1.570796, 1.398269],accel_mss,speed_ms,0,blend_radius_m)
    movel([-0.172737, -1.352660, -2.586154, -0.773575, 1.570796, 1.398059],accel_mss,speed_ms,0,blend_radius_m)
    movel([-0.173831, -1.347848, -2.589351, -0.775189, 1.570796, 1.396966],accel_mss,speed_ms,0,blend_radius_m)
    movel([-0.168773, -1.345194, -2.591101, -0.776093, 1.570796, 1.402023],accel_mss,speed_ms,0,blend_radius_m)
    movel([-0.169223, -1.343160, -2.592436, -0.776792, 1.570796, 1.401574],accel_mss,speed_ms,0,blend_radius_m)
    movel([-0.174292, -1.345828, -2.590684, -0.775876, 1.570796, 1.396505],accel_mss,speed_ms,0,blend_radius_m)
    movel([-0.175621, -1.340037, -2.594475, -0.777877, 1.570796, 1.395175],accel_mss,speed_ms,0,blend_radius_m)
    movel([-0.170518, -1.337328, -2.596232, -0.778829, 1.570796, 1.400279],accel_mss,speed_ms,0,blend_radius_m)
    movel([-0.171402, -1.333368, -2.598783, -0.780238, 1.570796, 1.399394],accel_mss,speed_ms,0,blend_radius_m)
    movel([-0.163769, -1.329319, -2.601369, -0.781700, 1.570796, 1.407028],accel_mss,speed_ms,0,blend_radius_m)
    movel([-0.162919, -1.333321, -2.598813, -0.780255, 1.570796, 1.407878],accel_mss,speed_ms,0,blend_radius_m)
    movel([-0.160246, -1.331919, -2.599711, -0.780759, 1.570796, 1.410551],accel_mss,speed_ms,0,blend_radius_m)
    movel([-0.161083, -1.327903, -2.602269, -0.782217, 1.570796, 1.409713],accel_mss,speed_ms,0,blend_radius_m)
    movel([-0.153386, -1.323865, -2.604819, -0.783706, 1.570796, 1.417410],accel_mss,speed_ms,0,blend_radius_m)
    movel([-0.152202, -1.329868, -2.601020, -0.781501, 1.570796, 1.418594],accel_mss,speed_ms,0,blend_radius_m)
    movel([-0.157369, -1.332552, -2.599306, -0.780531, 1.570796, 1.413427],accel_mss,speed_ms,0,blend_radius_m)
    movel([-0.156945, -1.334634, -2.597970, -0.779785, 1.570796, 1.413851],accel_mss,speed_ms,0,blend_radius_m)
    movel([-0.149106, -1.330580, -2.600566, -0.781243, 1.570796, 1.421690],accel_mss,speed_ms,0,blend_radius_m)
    movel([-0.150679, -1.322452, -2.605705, -0.784232, 1.570796, 1.420118],accel_mss,speed_ms,0,blend_radius_m)
    movel([-0.001924, -1.251119, -2.647144, -0.814126, 1.570796, 1.568873],accel_mss,speed_ms,0,blend_radius_m)
    speed_ms = 0.02
    movel([0.158957, -1.188696, -2.678386, -0.845308, 1.570796, 1.729754],accel_mss,speed_ms,0,blend_radius_m)
    movel([0.157034, -1.200160, -2.672976, -0.839253, 1.570796, 1.727831],accel_mss,speed_ms,0,blend_radius_m)
    speed_ms = 0.012
    movel([0.166189, -1.197160, -2.674405, -0.840823, 1.570796, 1.736986],accel_mss,speed_ms,0,blend_radius_m)
    movel([0.166716, -1.194184, -2.675814, -0.842391, 1.570796, 1.737513],accel_mss,speed_ms,0,blend_radius_m)
    movel([0.160669, -1.196167, -2.674876, -0.841345, 1.570796, 1.731466],accel_mss,speed_ms,0,blend_radius_m)
    movel([0.162134, -1.187639, -2.678877, -0.845873, 1.570796, 1.732930],accel_mss,speed_ms,0,blend_radius_m)
    movel([0.163603, -1.187149, -2.679104, -0.846136, 1.570796, 1.734399],accel_mss,speed_ms,0,blend_radius_m)
    movel([0.171178, -1.184645, -2.680263, -0.847481, 1.570796, 1.741974],accel_mss,speed_ms,0,blend_radius_m)
    movel([0.170131, -1.190457, -2.677564, -0.844368, 1.570796, 1.740927],accel_mss,speed_ms,0,blend_radius_m)
    movel([0.173284, -1.189438, -2.678039, -0.844911, 1.570796, 1.744080],accel_mss,speed_ms,0,blend_radius_m)
    movel([0.174358, -1.183606, -2.680741, -0.848041, 1.570796, 1.745154],accel_mss,speed_ms,0,blend_radius_m)
    movel([0.183424, -1.180682, -2.682083, -0.849624, 1.570796, 1.754220],accel_mss,speed_ms,0,blend_radius_m)
    movel([0.182294, -1.186557, -2.679379, -0.846453, 1.570796, 1.753091],accel_mss,speed_ms,0,blend_radius_m)
    movel([0.188385, -1.184641, -2.680265, -0.847483, 1.570796, 1.759181],accel_mss,speed_ms,0,blend_radius_m)
    movel([0.186680, -1.193280, -2.676240, -0.842870, 1.570796, 1.757477],accel_mss,speed_ms,0,blend_radius_m)
    movel([0.180648, -1.195154, -2.675356, -0.841879, 1.570796, 1.751444],accel_mss,speed_ms,0,blend_radius_m)
    movel([0.180078, -1.198139, -2.673940, -0.840310, 1.570796, 1.750875],accel_mss,speed_ms,0,blend_radius_m)
    movel([0.186090, -1.196283, -2.674822, -0.841285, 1.570796, 1.756886],accel_mss,speed_ms,0,blend_radius_m)
    movel([0.184696, -1.203394, -2.671424, -0.837571, 1.570796, 1.755493],accel_mss,speed_ms,0,blend_radius_m)
    movel([0.184428, -1.204765, -2.670763, -0.836861, 1.570796, 1.755225],accel_mss,speed_ms,0,blend_radius_m)
    movel([0.175610, -1.207468, -2.669453, -0.835468, 1.570796, 1.746407],accel_mss,speed_ms,0,blend_radius_m)
    movel([0.176673, -1.201793, -2.672194, -0.838402, 1.570796, 1.747469],accel_mss,speed_ms,0,blend_radius_m)
    movel([0.173563, -1.202767, -2.671726, -0.837896, 1.570796, 1.744359],accel_mss,speed_ms,0,blend_radius_m)
    movel([0.171983, -1.211350, -2.667557, -0.833482, 1.570796, 1.742780],accel_mss,speed_ms,0,blend_radius_m)
    movel([0.183853, -1.207714, -2.669333, -0.835342, 1.570796, 1.754649],accel_mss,speed_ms,0,blend_radius_m)
    speed_ms = 0.02
    movel([0.158243, -1.345021, -2.591215, -0.776152, 1.570796, 1.729039],accel_mss,speed_ms,0,blend_radius_m)
    movel([0.139022, -1.458254, -2.507595, -0.746540, 1.570796, 1.709818],accel_mss,speed_ms,0,blend_radius_m)
    speed_ms = 0.012
    movel([0.130132, -1.460164, -2.506021, -0.746204, 1.570796, 1.700928],accel_mss,speed_ms,0,blend_radius_m)
    movel([0.129256, -1.465966, -2.501205, -0.745218, 1.570796, 1.700052],accel_mss,speed_ms,0,blend_radius_m)
    movel([0.131545, -1.465473, -2.501616, -0.745300, 1.570796, 1.702341],accel_mss,speed_ms,0,blend_radius_m)
    movel([0.132131, -1.461656, -2.504788, -0.745945, 1.570796, 1.702927],accel_mss,speed_ms,0,blend_radius_m)
    movel([0.138690, -1.460258, -2.505944, -0.746187, 1.570796, 1.709487],accel_mss,speed_ms,0,blend_radius_m)
    movel([0.138542, -1.461182, -2.505180, -0.746027, 1.570796, 1.709338],accel_mss,speed_ms,0,blend_radius_m)
    movel([0.137780, -1.465926, -2.501239, -0.745225, 1.570796, 1.708576],accel_mss,speed_ms,0,blend_radius_m)
    movel([0.133380, -1.466851, -2.500465, -0.745072, 1.570796, 1.704177],accel_mss,speed_ms,0,blend_radius_m)
    movel([0.133075, -1.468822, -2.498815, -0.744752, 1.570796, 1.703871],accel_mss,speed_ms,0,blend_radius_m)
    movel([0.137466, -1.467900, -2.499588, -0.744901, 1.570796, 1.708263],accel_mss,speed_ms,0,blend_radius_m)
    movel([0.136570, -1.473508, -2.494867, -0.744014, 1.570796, 1.707367],accel_mss,speed_ms,0,blend_radius_m)
    speed_ms = 0.003
    movel([0.136570, -1.467543, -2.492148, -0.752698, 1.570796, 1.707367],accel_mss,speed_ms,0,blend_radius_m)
    speed_ms = 0.05
    movel([0.136570, -1.444454, -2.480985, -0.786951, 1.570796, 1.707367],accel_mss,speed_ms,0,blend_radius_m)
    #M_RunCode9
    movel([-0.101116, -1.322556, -2.569102, -0.820731, 1.570796, 1.469680],accel_mss,speed_ms,0,blend_radius_m)
    #M_RunCode3
    # num 0 inside
    movel([-0.101116, -1.347956, -2.581781, -0.782652, 1.570796, 1.469680],accel_mss,speed_ms,0,blend_radius_m)
    speed_ms = 0.003
    movel([-0.101116, -1.354564, -2.584879, -0.772945, 1.570796, 1.469680],accel_mss,speed_ms,0,blend_radius_m)
    speed_ms = 0.015
    movel([-0.106161, -1.361335, -2.580307, -0.770747, 1.570796, 1.464635],accel_mss,speed_ms,0,blend_radius_m)
    movel([-0.110090, -1.365943, -2.577159, -0.769287, 1.570796, 1.460707],accel_mss,speed_ms,0,blend_radius_m)
    movel([-0.111700, -1.367455, -2.576119, -0.768814, 1.570796, 1.459096],accel_mss,speed_ms,0,blend_radius_m)
    movel([-0.113150, -1.368443, -2.575438, -0.768507, 1.570796, 1.457647],accel_mss,speed_ms,0,blend_radius_m)
    movel([-0.114438, -1.368913, -2.575114, -0.768362, 1.570796, 1.456358],accel_mss,speed_ms,0,blend_radius_m)
    movel([-0.115571, -1.368864, -2.575148, -0.768377, 1.570796, 1.455226],accel_mss,speed_ms,0,blend_radius_m)
    movel([-0.116374, -1.368348, -2.575504, -0.768537, 1.570796, 1.454422],accel_mss,speed_ms,0,blend_radius_m)
    movel([-0.116674, -1.367414, -2.576148, -0.768827, 1.570796, 1.454122],accel_mss,speed_ms,0,blend_radius_m)
    movel([-0.116470, -1.366059, -2.577080, -0.769251, 1.570796, 1.454326],accel_mss,speed_ms,0,blend_radius_m)
    movel([-0.115761, -1.364279, -2.578299, -0.769810, 1.570796, 1.455035],accel_mss,speed_ms,0,blend_radius_m)
    movel([-0.112933, -1.359327, -2.581670, -0.771392, 1.570796, 1.457863],accel_mss,speed_ms,0,blend_radius_m)
    movel([-0.108281, -1.352413, -2.586319, -0.773657, 1.570796, 1.462515],accel_mss,speed_ms,0,blend_radius_m)
    movel([-0.103194, -1.345531, -2.590880, -0.775978, 1.570796, 1.467603],accel_mss,speed_ms,0,blend_radius_m)
    movel([-0.099141, -1.340763, -2.594002, -0.777624, 1.570796, 1.471655],accel_mss,speed_ms,0,blend_radius_m)
    movel([-0.097464, -1.339187, -2.595027, -0.778175, 1.570796, 1.473333],accel_mss,speed_ms,0,blend_radius_m)
    movel([-0.095957, -1.338153, -2.595698, -0.778538, 1.570796, 1.474840],accel_mss,speed_ms,0,blend_radius_m)
    movel([-0.094620, -1.337665, -2.596014, -0.778710, 1.570796, 1.476176],accel_mss,speed_ms,0,blend_radius_m)
    movel([-0.093457, -1.337724, -2.595976, -0.778689, 1.570796, 1.477339],accel_mss,speed_ms,0,blend_radius_m)
    movel([-0.092647, -1.338276, -2.595618, -0.778495, 1.570796, 1.478149],accel_mss,speed_ms,0,blend_radius_m)
    movel([-0.092365, -1.339263, -2.594978, -0.778148, 1.570796, 1.478432],accel_mss,speed_ms,0,blend_radius_m)
    movel([-0.092614, -1.340685, -2.594053, -0.777651, 1.570796, 1.478183],accel_mss,speed_ms,0,blend_radius_m)
    movel([-0.093386, -1.342532, -2.592847, -0.777009, 1.570796, 1.477410],accel_mss,speed_ms,0,blend_radius_m)
    movel([-0.096363, -1.347612, -2.589507, -0.775269, 1.570796, 1.474433],accel_mss,speed_ms,0,blend_radius_m)
    movel([-0.101116, -1.354564, -2.584879, -0.772945, 1.570796, 1.469680],accel_mss,speed_ms,0,blend_radius_m)
    speed_ms = 0.003
    movel([-0.101116, -1.347956, -2.581781, -0.782652, 1.570796, 1.469680],accel_mss,speed_ms,0,blend_radius_m)
    speed_ms = 0.05
    movel([-0.101116, -1.322556, -2.569102, -0.820731, 1.570796, 1.469680],accel_mss,speed_ms,0,blend_radius_m)
    #M_RunCode9
    movel([-0.093439, -1.325002, -2.567533, -0.819854, 1.570796, 1.477357],accel_mss,speed_ms,0,blend_radius_m)
    #M_RunCode3
    #num 0 outside
    movel([-0.093439, -1.350361, -2.580180, -0.781848, 1.570796, 1.477357],accel_mss,speed_ms,0,blend_radius_m)
    speed_ms = 0.003
    movel([-0.093439, -1.356958, -2.583270, -0.772161, 1.570796, 1.477357],accel_mss,speed_ms,0,blend_radius_m)
    speed_ms = 0.015
    movel([-0.095323, -1.359406, -2.581617, -0.771367, 1.570796, 1.475474],accel_mss,speed_ms,0,blend_radius_m)
    movel([-0.097250, -1.361605, -2.580124, -0.770660, 1.570796, 1.473546],accel_mss,speed_ms,0,blend_radius_m)
    movel([-0.099225, -1.363562, -2.578790, -0.770037, 1.570796, 1.471571],accel_mss,speed_ms,0,blend_radius_m)
    movel([-0.101247, -1.365276, -2.577617, -0.769496, 1.570796, 1.469549],accel_mss,speed_ms,0,blend_radius_m)
    movel([-0.103277, -1.366737, -2.576613, -0.769038, 1.570796, 1.467519],accel_mss,speed_ms,0,blend_radius_m)
    movel([-0.105274, -1.367936, -2.575788, -0.768665, 1.570796, 1.465522],accel_mss,speed_ms,0,blend_radius_m)
    movel([-0.107241, -1.368876, -2.575140, -0.768373, 1.570796, 1.463555],accel_mss,speed_ms,0,blend_radius_m)
    movel([-0.109177, -1.369553, -2.574672, -0.768164, 1.570796, 1.461619],accel_mss,speed_ms,0,blend_radius_m)
    movel([-0.111057, -1.369973, -2.574381, -0.768035, 1.570796, 1.459739],accel_mss,speed_ms,0,blend_radius_m)
    movel([-0.112847, -1.370143, -2.574264, -0.767982, 1.570796, 1.457949],accel_mss,speed_ms,0,blend_radius_m)
    movel([-0.114554, -1.370059, -2.574322, -0.768008, 1.570796, 1.456243],accel_mss,speed_ms,0,blend_radius_m)
    movel([-0.116176, -1.369726, -2.574552, -0.768111, 1.570796, 1.454621],accel_mss,speed_ms,0,blend_radius_m)
    movel([-0.117639, -1.369161, -2.574943, -0.768285, 1.570796, 1.453158],accel_mss,speed_ms,0,blend_radius_m)
    movel([-0.118861, -1.368389, -2.575476, -0.768524, 1.570796, 1.451935],accel_mss,speed_ms,0,blend_radius_m)
    movel([-0.119847, -1.367410, -2.576151, -0.768828, 1.570796, 1.450949],accel_mss,speed_ms,0,blend_radius_m)
    movel([-0.120593, -1.366216, -2.576972, -0.769201, 1.570796, 1.450203],accel_mss,speed_ms,0,blend_radius_m)
    movel([-0.121076, -1.364824, -2.577927, -0.769639, 1.570796, 1.449720],accel_mss,speed_ms,0,blend_radius_m)
    movel([-0.121271, -1.363244, -2.579007, -0.770138, 1.570796, 1.449525],accel_mss,speed_ms,0,blend_radius_m)
    movel([-0.121177, -1.361471, -2.580215, -0.770703, 1.570796, 1.449619],accel_mss,speed_ms,0,blend_radius_m)
    movel([-0.120789, -1.359505, -2.581549, -0.771335, 1.570796, 1.450007],accel_mss,speed_ms,0,blend_radius_m)
    movel([-0.120098, -1.357373, -2.582991, -0.772026, 1.570796, 1.450698],accel_mss,speed_ms,0,blend_radius_m)
    movel([-0.119085, -1.355103, -2.584518, -0.772768, 1.570796, 1.451711],accel_mss,speed_ms,0,blend_radius_m)
    movel([-0.117751, -1.352697, -2.586129, -0.773563, 1.570796, 1.453045],accel_mss,speed_ms,0,blend_radius_m)
    movel([-0.116093, -1.350152, -2.587824, -0.774413, 1.570796, 1.454704],accel_mss,speed_ms,0,blend_radius_m)
    movel([-0.114233, -1.347648, -2.589484, -0.775257, 1.570796, 1.456564],accel_mss,speed_ms,0,blend_radius_m)
    movel([-0.112304, -1.345376, -2.590982, -0.776031, 1.570796, 1.458493],accel_mss,speed_ms,0,blend_radius_m)
    movel([-0.110305, -1.343337, -2.592320, -0.776731, 1.570796, 1.460492],accel_mss,speed_ms,0,blend_radius_m)
    movel([-0.108239, -1.341537, -2.593498, -0.777355, 1.570796, 1.462557],accel_mss,speed_ms,0,blend_radius_m)
    movel([-0.106152, -1.339991, -2.594504, -0.777893, 1.570796, 1.464644],accel_mss,speed_ms,0,blend_radius_m)
    movel([-0.104092, -1.338723, -2.595328, -0.778337, 1.570796, 1.466704],accel_mss,speed_ms,0,blend_radius_m)
    movel([-0.102059, -1.337730, -2.595972, -0.778687, 1.570796, 1.468737],accel_mss,speed_ms,0,blend_radius_m)
    movel([-0.100055, -1.337017, -2.596433, -0.778939, 1.570796, 1.470741],accel_mss,speed_ms,0,blend_radius_m)
    movel([-0.098115, -1.336579, -2.596716, -0.779094, 1.570796, 1.472681],accel_mss,speed_ms,0,blend_radius_m)
    movel([-0.096266, -1.336409, -2.596826, -0.779154, 1.570796, 1.474530],accel_mss,speed_ms,0,blend_radius_m)
    movel([-0.094508, -1.336506, -2.596763, -0.779120, 1.570796, 1.476288],accel_mss,speed_ms,0,blend_radius_m)
    movel([-0.092848, -1.336874, -2.596526, -0.778989, 1.570796, 1.477948],accel_mss,speed_ms,0,blend_radius_m)
    movel([-0.091363, -1.337486, -2.596130, -0.778773, 1.570796, 1.479434],accel_mss,speed_ms,0,blend_radius_m)
    movel([-0.090132, -1.338313, -2.595594, -0.778482, 1.570796, 1.480664],accel_mss,speed_ms,0,blend_radius_m)
    movel([-0.089156, -1.339357, -2.594917, -0.778115, 1.570796, 1.481641],accel_mss,speed_ms,0,blend_radius_m)
    movel([-0.088434, -1.340616, -2.594098, -0.777675, 1.570796, 1.482363],accel_mss,speed_ms,0,blend_radius_m)
    movel([-0.087990, -1.342075, -2.593146, -0.777168, 1.570796, 1.482806],accel_mss,speed_ms,0,blend_radius_m)
    movel([-0.087851, -1.343724, -2.592067, -0.776598, 1.570796, 1.482946],accel_mss,speed_ms,0,blend_radius_m)
    movel([-0.088015, -1.345563, -2.590859, -0.775967, 1.570796, 1.482781],accel_mss,speed_ms,0,blend_radius_m)
    movel([-0.088479, -1.347585, -2.589526, -0.775279, 1.570796, 1.482317],accel_mss,speed_ms,0,blend_radius_m)
    movel([-0.089250, -1.349756, -2.588088, -0.774546, 1.570796, 1.481546],accel_mss,speed_ms,0,blend_radius_m)
    movel([-0.090337, -1.352044, -2.586565, -0.773780, 1.570796, 1.480459],accel_mss,speed_ms,0,blend_radius_m)
    movel([-0.091734, -1.354445, -2.584959, -0.772985, 1.570796, 1.479062],accel_mss,speed_ms,0,blend_radius_m)
    movel([-0.093439, -1.356958, -2.583270, -0.772161, 1.570796, 1.477357],accel_mss,speed_ms,0,blend_radius_m)
    speed_ms = 0.003
    movel([-0.093439, -1.350361, -2.580180, -0.781848, 1.570796, 1.477357],accel_mss,speed_ms,0,blend_radius_m)
    speed_ms = 0.05
    movel([-0.093439, -1.325002, -2.567533, -0.819854, 1.570796, 1.477357],accel_mss,speed_ms,0,blend_radius_m)
    #M_RunCode9
    movel([-0.123954, -1.324456, -2.567884, -0.820049, 1.570796, 1.446843],accel_mss,speed_ms,0,blend_radius_m)
    #M_RunCode3
    # num 2
    movel([-0.123954, -1.349824, -2.580538, -0.782027, 1.570796, 1.446843],accel_mss,speed_ms,0,blend_radius_m)
    speed_ms = 0.003
    movel([-0.123954, -1.356423, -2.583630, -0.772335, 1.570796, 1.446843],accel_mss,speed_ms,0,blend_radius_m)
    speed_ms = 0.02
    movel([-0.129998, -1.365194, -2.577673, -0.769522, 1.570796, 1.440798],accel_mss,speed_ms,0,blend_radius_m)
    movel([-0.153716, -1.359168, -2.581778, -0.771443, 1.570796, 1.417080],accel_mss,speed_ms,0,blend_radius_m)
    movel([-0.153133, -1.358284, -2.582375, -0.771729, 1.570796, 1.417664],accel_mss,speed_ms,0,blend_radius_m)
    movel([-0.151367, -1.356095, -2.583852, -0.772443, 1.570796, 1.419429],accel_mss,speed_ms,0,blend_radius_m)
    movel([-0.149072, -1.354075, -2.585207, -0.773107, 1.570796, 1.421725],accel_mss,speed_ms,0,blend_radius_m)
    movel([-0.146447, -1.352249, -2.586428, -0.773712, 1.570796, 1.424349],accel_mss,speed_ms,0,blend_radius_m)
    movel([-0.143702, -1.350644, -2.587497, -0.774248, 1.570796, 1.427094],accel_mss,speed_ms,0,blend_radius_m)
    movel([-0.136140, -1.346869, -2.589998, -0.775522, 1.570796, 1.434656],accel_mss,speed_ms,0,blend_radius_m)
    movel([-0.129079, -1.343432, -2.592258, -0.776699, 1.570796, 1.441717],accel_mss,speed_ms,0,blend_radius_m)
    movel([-0.126471, -1.341951, -2.593227, -0.777211, 1.570796, 1.444325],accel_mss,speed_ms,0,blend_radius_m)
    movel([-0.124017, -1.340294, -2.594308, -0.777788, 1.570796, 1.446780],accel_mss,speed_ms,0,blend_radius_m)
    movel([-0.121890, -1.338487, -2.595482, -0.778421, 1.570796, 1.448906],accel_mss,speed_ms,0,blend_radius_m)
    movel([-0.120264, -1.336553, -2.596733, -0.779103, 1.570796, 1.450532],accel_mss,speed_ms,0,blend_radius_m)
    movel([-0.118963, -1.334098, -2.598315, -0.779977, 1.570796, 1.451833],accel_mss,speed_ms,0,blend_radius_m)
    movel([-0.118722, -1.333042, -2.598992, -0.780355, 1.570796, 1.452075],accel_mss,speed_ms,0,blend_radius_m)
    movel([-0.118753, -1.332102, -2.599594, -0.780693, 1.570796, 1.452044],accel_mss,speed_ms,0,blend_radius_m)
    movel([-0.119446, -1.330656, -2.600518, -0.781215, 1.570796, 1.451350],accel_mss,speed_ms,0,blend_radius_m)
    movel([-0.120855, -1.329858, -2.601026, -0.781505, 1.570796, 1.449941],accel_mss,speed_ms,0,blend_radius_m)
    movel([-0.122064, -1.329696, -2.601129, -0.781563, 1.570796, 1.448732],accel_mss,speed_ms,0,blend_radius_m)
    movel([-0.123171, -1.329886, -2.601009, -0.781495, 1.570796, 1.447625],accel_mss,speed_ms,0,blend_radius_m)
    movel([-0.124102, -1.330365, -2.600703, -0.781321, 1.570796, 1.446695],accel_mss,speed_ms,0,blend_radius_m)
    movel([-0.124778, -1.331064, -2.600258, -0.781068, 1.570796, 1.446018],accel_mss,speed_ms,0,blend_radius_m)
    movel([-0.125119, -1.332265, -2.599490, -0.780634, 1.570796, 1.445678],accel_mss,speed_ms,0,blend_radius_m)
    movel([-0.125345, -1.333426, -2.598746, -0.780217, 1.570796, 1.445451],accel_mss,speed_ms,0,blend_radius_m)
    movel([-0.126105, -1.334850, -2.597831, -0.779708, 1.570796, 1.444691],accel_mss,speed_ms,0,blend_radius_m)
    movel([-0.127495, -1.336400, -2.596832, -0.779157, 1.570796, 1.443301],accel_mss,speed_ms,0,blend_radius_m)
    movel([-0.129163, -1.337385, -2.596195, -0.778809, 1.570796, 1.441634],accel_mss,speed_ms,0,blend_radius_m)
    movel([-0.130909, -1.337812, -2.595919, -0.778658, 1.570796, 1.439887],accel_mss,speed_ms,0,blend_radius_m)
    movel([-0.132535, -1.337687, -2.596000, -0.778702, 1.570796, 1.438262],accel_mss,speed_ms,0,blend_radius_m)
    movel([-0.133822, -1.337065, -2.596402, -0.778922, 1.570796, 1.436975],accel_mss,speed_ms,0,blend_radius_m)
    movel([-0.134561, -1.335997, -2.597092, -0.779300, 1.570796, 1.436235],accel_mss,speed_ms,0,blend_radius_m)
    movel([-0.134602, -1.334568, -2.598012, -0.779809, 1.570796, 1.436194],accel_mss,speed_ms,0,blend_radius_m)
    movel([-0.133790, -1.332863, -2.599107, -0.780419, 1.570796, 1.437007],accel_mss,speed_ms,0,blend_radius_m)
    movel([-0.132656, -1.331465, -2.600001, -0.780923, 1.570796, 1.438141],accel_mss,speed_ms,0,blend_radius_m)
    movel([-0.131309, -1.330326, -2.600728, -0.781335, 1.570796, 1.439487],accel_mss,speed_ms,0,blend_radius_m)
    movel([-0.129748, -1.329445, -2.601289, -0.781655, 1.570796, 1.441048],accel_mss,speed_ms,0,blend_radius_m)
    movel([-0.127974, -1.328829, -2.601681, -0.781879, 1.570796, 1.442823],accel_mss,speed_ms,0,blend_radius_m)
    movel([-0.126079, -1.328474, -2.601907, -0.782009, 1.570796, 1.444717],accel_mss,speed_ms,0,blend_radius_m)
    movel([-0.124154, -1.328370, -2.601972, -0.782047, 1.570796, 1.446642],accel_mss,speed_ms,0,blend_radius_m)
    movel([-0.120221, -1.328934, -2.601614, -0.781841, 1.570796, 1.450575],accel_mss,speed_ms,0,blend_radius_m)
    movel([-0.117965, -1.329713, -2.601118, -0.781557, 1.570796, 1.452832],accel_mss,speed_ms,0,blend_radius_m)
    movel([-0.116035, -1.330744, -2.600461, -0.781183, 1.570796, 1.454762],accel_mss,speed_ms,0,blend_radius_m)
    movel([-0.114434, -1.332023, -2.599645, -0.780721, 1.570796, 1.456362],accel_mss,speed_ms,0,blend_radius_m)
    movel([-0.113162, -1.333549, -2.598667, -0.780173, 1.570796, 1.457634],accel_mss,speed_ms,0,blend_radius_m)
    movel([-0.112422, -1.335319, -2.597529, -0.779541, 1.570796, 1.458375],accel_mss,speed_ms,0,blend_radius_m)
    movel([-0.112423, -1.337340, -2.596224, -0.778825, 1.570796, 1.458373],accel_mss,speed_ms,0,blend_radius_m)
    movel([-0.113159, -1.339605, -2.594755, -0.778028, 1.570796, 1.457637],accel_mss,speed_ms,0,blend_radius_m)
    movel([-0.114621, -1.342110, -2.593123, -0.777156, 1.570796, 1.456175],accel_mss,speed_ms,0,blend_radius_m)
    movel([-0.116384, -1.344285, -2.591699, -0.776405, 1.570796, 1.454412],accel_mss,speed_ms,0,blend_radius_m)
    movel([-0.118449, -1.346179, -2.590453, -0.775757, 1.570796, 1.452347],accel_mss,speed_ms,0,blend_radius_m)
    movel([-0.120701, -1.347816, -2.589373, -0.775200, 1.570796, 1.450095],accel_mss,speed_ms,0,blend_radius_m)
    movel([-0.123019, -1.349217, -2.588445, -0.774727, 1.570796, 1.447777],accel_mss,speed_ms,0,blend_radius_m)
    movel([-0.128882, -1.352127, -2.586509, -0.773752, 1.570796, 1.441914],accel_mss,speed_ms,0,blend_radius_m)
    movel([-0.134390, -1.354902, -2.584653, -0.772834, 1.570796, 1.436406],accel_mss,speed_ms,0,blend_radius_m)
    movel([-0.136479, -1.356170, -2.583801, -0.772418, 1.570796, 1.434317],accel_mss,speed_ms,0,blend_radius_m)
    movel([-0.138470, -1.357620, -2.582824, -0.771945, 1.570796, 1.432326],accel_mss,speed_ms,0,blend_radius_m)
    movel([-0.140252, -1.359262, -2.581714, -0.771413, 1.570796, 1.430544],accel_mss,speed_ms,0,blend_radius_m)
    movel([-0.141709, -1.361091, -2.580474, -0.770825, 1.570796, 1.429087],accel_mss,speed_ms,0,blend_radius_m)
    movel([-0.140820, -1.361317, -2.580320, -0.770752, 1.570796, 1.429976],accel_mss,speed_ms,0,blend_radius_m)
    movel([-0.138271, -1.361815, -2.579981, -0.770593, 1.570796, 1.432526],accel_mss,speed_ms,0,blend_radius_m)
    movel([-0.135841, -1.361968, -2.579877, -0.770544, 1.570796, 1.434956],accel_mss,speed_ms,0,blend_radius_m)
    movel([-0.133532, -1.361779, -2.580005, -0.770605, 1.570796, 1.437265],accel_mss,speed_ms,0,blend_radius_m)
    movel([-0.131335, -1.361242, -2.580371, -0.770776, 1.570796, 1.439461],accel_mss,speed_ms,0,blend_radius_m)
    movel([-0.129273, -1.360410, -2.580936, -0.771043, 1.570796, 1.441523],accel_mss,speed_ms,0,blend_radius_m)
    movel([-0.127356, -1.359331, -2.581667, -0.771391, 1.570796, 1.443441],accel_mss,speed_ms,0,blend_radius_m)
    movel([-0.125585, -1.358004, -2.582565, -0.771820, 1.570796, 1.445212],accel_mss,speed_ms,0,blend_radius_m)
    movel([-0.123954, -1.356423, -2.583630, -0.772335, 1.570796, 1.446843],accel_mss,speed_ms,0,blend_radius_m)
    speed_ms = 0.003
    movel([-0.123954, -1.349824, -2.580538, -0.782027, 1.570796, 1.446843],accel_mss,speed_ms,0,blend_radius_m)
    speed_ms = 0.05
    movel([-0.123954, -1.324456, -2.567884, -0.820049, 1.570796, 1.446843],accel_mss,speed_ms,0,blend_radius_m)
    #M_RunCode9
    movel([0.068760, -1.419496, -2.500728, -0.792166, 1.570796, 1.639556],accel_mss,speed_ms,0,blend_radius_m)
    #M_RunCode3
    movel([0.068760, -1.443093, -2.512190, -0.757106, 1.570796, 1.639556],accel_mss,speed_ms,0,blend_radius_m)
    speed_ms = 0.003
    movel([0.068760, -1.449197, -2.514984, -0.748208, 1.570796, 1.639556],accel_mss,speed_ms,0,blend_radius_m)
    speed_ms = 0.02
    movel([0.070663, -1.447541, -2.516321, -0.748527, 1.570796, 1.641460],accel_mss,speed_ms,0,blend_radius_m)
    movel([0.072941, -1.446164, -2.517430, -0.748795, 1.570796, 1.643737],accel_mss,speed_ms,0,blend_radius_m)
    movel([0.075428, -1.445044, -2.518330, -0.749016, 1.570796, 1.646225],accel_mss,speed_ms,0,blend_radius_m)
    movel([0.077955, -1.444162, -2.519036, -0.749190, 1.570796, 1.648751],accel_mss,speed_ms,0,blend_radius_m)
    movel([0.084751, -1.442342, -2.520492, -0.749555, 1.570796, 1.655547],accel_mss,speed_ms,0,blend_radius_m)
    movel([0.091060, -1.440730, -2.521777, -0.749882, 1.570796, 1.661856],accel_mss,speed_ms,0,blend_radius_m)
    movel([0.093434, -1.439943, -2.522403, -0.750043, 1.570796, 1.664230],accel_mss,speed_ms,0,blend_radius_m)
    movel([0.095728, -1.438957, -2.523186, -0.750246, 1.570796, 1.666524],accel_mss,speed_ms,0,blend_radius_m)
    movel([0.097799, -1.437760, -2.524135, -0.750494, 1.570796, 1.668595],accel_mss,speed_ms,0,blend_radius_m)
    movel([0.099508, -1.436334, -2.525261, -0.750793, 1.570796, 1.670304],accel_mss,speed_ms,0,blend_radius_m)
    movel([0.101083, -1.434354, -2.526822, -0.751213, 1.570796, 1.671879],accel_mss,speed_ms,0,blend_radius_m)
    movel([0.101514, -1.433430, -2.527547, -0.751411, 1.570796, 1.672310],accel_mss,speed_ms,0,blend_radius_m)
    movel([0.101707, -1.432553, -2.528235, -0.751601, 1.570796, 1.672503],accel_mss,speed_ms,0,blend_radius_m)
    movel([0.101503, -1.431056, -2.529407, -0.751926, 1.570796, 1.672299],accel_mss,speed_ms,0,blend_radius_m)
    movel([0.100596, -1.429995, -2.530235, -0.752159, 1.570796, 1.671393],accel_mss,speed_ms,0,blend_radius_m)
    movel([0.099697, -1.429566, -2.530569, -0.752254, 1.570796, 1.670494],accel_mss,speed_ms,0,blend_radius_m)
    movel([0.098793, -1.429491, -2.530627, -0.752270, 1.570796, 1.669589],accel_mss,speed_ms,0,blend_radius_m)
    movel([0.097963, -1.429720, -2.530449, -0.752220, 1.570796, 1.668759],accel_mss,speed_ms,0,blend_radius_m)
    movel([0.097276, -1.430214, -2.530064, -0.752111, 1.570796, 1.668072],accel_mss,speed_ms,0,blend_radius_m)
    movel([0.096732, -1.431251, -2.529254, -0.751884, 1.570796, 1.667529],accel_mss,speed_ms,0,blend_radius_m)
    movel([0.096287, -1.432279, -2.528450, -0.751660, 1.570796, 1.667083],accel_mss,speed_ms,0,blend_radius_m)
    movel([0.095363, -1.433428, -2.527549, -0.751412, 1.570796, 1.666159],accel_mss,speed_ms,0,blend_radius_m)
    movel([0.093925, -1.434552, -2.526666, -0.751171, 1.570796, 1.664721],accel_mss,speed_ms,0,blend_radius_m)
    movel([0.092399, -1.435087, -2.526245, -0.751057, 1.570796, 1.663196],accel_mss,speed_ms,0,blend_radius_m)
    movel([0.090939, -1.435088, -2.526244, -0.751057, 1.570796, 1.661735],accel_mss,speed_ms,0,blend_radius_m)
    movel([0.089706, -1.434602, -2.526627, -0.751160, 1.570796, 1.660503],accel_mss,speed_ms,0,blend_radius_m)
    movel([0.088851, -1.433727, -2.527315, -0.751348, 1.570796, 1.659647],accel_mss,speed_ms,0,blend_radius_m)
    movel([0.088526, -1.432563, -2.528227, -0.751598, 1.570796, 1.659322],accel_mss,speed_ms,0,blend_radius_m)
    movel([0.088829, -1.431224, -2.529275, -0.751890, 1.570796, 1.659626],accel_mss,speed_ms,0,blend_radius_m)
    movel([0.089862, -1.429823, -2.530369, -0.752197, 1.570796, 1.660658],accel_mss,speed_ms,0,blend_radius_m)
    movel([0.091068, -1.428780, -2.531181, -0.752428, 1.570796, 1.661865],accel_mss,speed_ms,0,blend_radius_m)
    movel([0.092383, -1.428029, -2.531765, -0.752595, 1.570796, 1.663180],accel_mss,speed_ms,0,blend_radius_m)
    movel([0.093800, -1.427571, -2.532121, -0.752697, 1.570796, 1.664596],accel_mss,speed_ms,0,blend_radius_m)
    movel([0.095318, -1.427407, -2.532248, -0.752734, 1.570796, 1.666114],accel_mss,speed_ms,0,blend_radius_m)
    movel([0.096869, -1.427511, -2.532167, -0.752711, 1.570796, 1.667665],accel_mss,speed_ms,0,blend_radius_m)
    movel([0.098384, -1.427860, -2.531896, -0.752633, 1.570796, 1.669180],accel_mss,speed_ms,0,blend_radius_m)
    movel([0.101302, -1.429281, -2.530791, -0.752317, 1.570796, 1.672098],accel_mss,speed_ms,0,blend_radius_m)
    movel([0.102869, -1.430520, -2.529825, -0.752044, 1.570796, 1.673665],accel_mss,speed_ms,0,blend_radius_m)
    movel([0.104126, -1.431914, -2.528736, -0.751739, 1.570796, 1.674922],accel_mss,speed_ms,0,blend_radius_m)
    movel([0.105072, -1.433460, -2.527524, -0.751405, 1.570796, 1.675868],accel_mss,speed_ms,0,blend_radius_m)
    movel([0.105708, -1.435158, -2.526189, -0.751042, 1.570796, 1.676504],accel_mss,speed_ms,0,blend_radius_m)
    movel([0.105875, -1.436962, -2.524766, -0.750661, 1.570796, 1.676672],accel_mss,speed_ms,0,blend_radius_m)
    movel([0.105413, -1.438830, -2.523287, -0.750272, 1.570796, 1.676209],accel_mss,speed_ms,0,blend_radius_m)
    movel([0.104327, -1.440758, -2.521755, -0.749876, 1.570796, 1.675124],accel_mss,speed_ms,0,blend_radius_m)
    movel([0.102618, -1.442749, -2.520167, -0.749473, 1.570796, 1.673414],accel_mss,speed_ms,0,blend_radius_m)
    movel([0.100753, -1.444369, -2.518871, -0.749149, 1.570796, 1.671549],accel_mss,speed_ms,0,blend_radius_m)
    movel([0.098712, -1.445664, -2.517832, -0.748893, 1.570796, 1.669508],accel_mss,speed_ms,0,blend_radius_m)
    movel([0.096580, -1.446682, -2.517013, -0.748694, 1.570796, 1.667376],accel_mss,speed_ms,0,blend_radius_m)
    movel([0.094453, -1.447465, -2.516382, -0.748542, 1.570796, 1.665249],accel_mss,speed_ms,0,blend_radius_m)
    movel([0.089204, -1.448866, -2.515251, -0.748272, 1.570796, 1.660000],accel_mss,speed_ms,0,blend_radius_m)
    movel([0.084253, -1.450226, -2.514150, -0.748013, 1.570796, 1.655049],accel_mss,speed_ms,0,blend_radius_m)
    movel([0.082323, -1.450941, -2.513570, -0.747877, 1.570796, 1.653120],accel_mss,speed_ms,0,blend_radius_m)
    movel([0.080426, -1.451855, -2.512828, -0.747706, 1.570796, 1.651222],accel_mss,speed_ms,0,blend_radius_m)
    movel([0.078646, -1.452992, -2.511903, -0.747494, 1.570796, 1.649443],accel_mss,speed_ms,0,blend_radius_m)
    movel([0.077077, -1.454379, -2.510772, -0.747238, 1.570796, 1.647873],accel_mss,speed_ms,0,blend_radius_m)
    movel([0.077721, -1.454788, -2.510438, -0.747163, 1.570796, 1.648517],accel_mss,speed_ms,0,blend_radius_m)
    movel([0.079611, -1.455815, -2.509597, -0.746977, 1.570796, 1.650407],accel_mss,speed_ms,0,blend_radius_m)
    movel([0.081484, -1.456496, -2.509039, -0.746854, 1.570796, 1.652280],accel_mss,speed_ms,0,blend_radius_m)
    movel([0.083340, -1.456829, -2.508766, -0.746794, 1.570796, 1.654136],accel_mss,speed_ms,0,blend_radius_m)
    movel([0.085185, -1.456812, -2.508780, -0.746797, 1.570796, 1.655981],accel_mss,speed_ms,0,blend_radius_m)
    movel([0.086996, -1.456490, -2.509044, -0.746855, 1.570796, 1.657792],accel_mss,speed_ms,0,blend_radius_m)
    movel([0.088744, -1.455908, -2.509521, -0.746960, 1.570796, 1.659540],accel_mss,speed_ms,0,blend_radius_m)
    movel([0.090437, -1.455062, -2.510213, -0.747113, 1.570796, 1.661233],accel_mss,speed_ms,0,blend_radius_m)
    movel([0.092073, -1.453953, -2.511120, -0.747317, 1.570796, 1.662869],accel_mss,speed_ms,0,blend_radius_m)
    movel([0.085333, -1.460787, -2.505507, -0.746096, 1.570796, 1.656129],accel_mss,speed_ms,0,blend_radius_m)
    movel([0.068092, -1.449897, -2.514417, -0.748075, 1.570796, 1.638889],accel_mss,speed_ms,0,blend_radius_m)
    movel([0.068760, -1.449197, -2.514984, -0.748208, 1.570796, 1.639556],accel_mss,speed_ms,0,blend_radius_m)
    speed_ms = 0.003
    movel([0.068760, -1.443093, -2.512190, -0.757106, 1.570796, 1.639556],accel_mss,speed_ms,0,blend_radius_m)
    speed_ms = 0.05
    movel([0.068760, -1.419496, -2.500728, -0.792166, 1.570796, 1.639556],accel_mss,speed_ms,0,blend_radius_m)
    #M_RunCode9
    movel([0.091644, -1.428444, -2.493753, -0.790192, 1.570796, 1.662440],accel_mss,speed_ms,0,blend_radius_m)
    #M_RunCode3
    movel([0.091644, -1.451861, -2.505107, -0.755421, 1.570796, 1.662440],accel_mss,speed_ms,0,blend_radius_m)
    speed_ms = 0.003
    movel([0.091644, -1.457915, -2.507874, -0.746600, 1.570796, 1.662440],accel_mss,speed_ms,0,blend_radius_m)
    speed_ms = 0.02
    movel([0.093047, -1.456830, -2.508765, -0.746794, 1.570796, 1.663844],accel_mss,speed_ms,0,blend_radius_m)
    movel([0.094548, -1.456307, -2.509194, -0.746888, 1.570796, 1.665344],accel_mss,speed_ms,0,blend_radius_m)
    movel([0.095984, -1.456307, -2.509194, -0.746888, 1.570796, 1.666781],accel_mss,speed_ms,0,blend_radius_m)
    movel([0.097185, -1.456794, -2.508795, -0.746800, 1.570796, 1.667982],accel_mss,speed_ms,0,blend_radius_m)
    movel([0.098001, -1.457663, -2.508081, -0.746645, 1.570796, 1.668797],accel_mss,speed_ms,0,blend_radius_m)
    movel([0.098284, -1.458816, -2.507133, -0.746440, 1.570796, 1.669081],accel_mss,speed_ms,0,blend_radius_m)
    movel([0.097962, -1.460123, -2.506055, -0.746211, 1.570796, 1.668759],accel_mss,speed_ms,0,blend_radius_m)
    movel([0.096952, -1.461458, -2.504951, -0.745979, 1.570796, 1.667749],accel_mss,speed_ms,0,blend_radius_m)
    movel([0.095818, -1.462389, -2.504180, -0.745820, 1.570796, 1.666614],accel_mss,speed_ms,0,blend_radius_m)
    movel([0.094731, -1.462927, -2.503734, -0.745728, 1.570796, 1.665527],accel_mss,speed_ms,0,blend_radius_m)
    movel([0.093654, -1.463543, -2.503222, -0.745623, 1.570796, 1.664451],accel_mss,speed_ms,0,blend_radius_m)
    movel([0.093235, -1.464167, -2.502704, -0.745518, 1.570796, 1.664031],accel_mss,speed_ms,0,blend_radius_m)
    movel([0.093155, -1.464858, -2.502129, -0.745402, 1.570796, 1.663951],accel_mss,speed_ms,0,blend_radius_m)
    movel([0.093385, -1.465511, -2.501584, -0.745293, 1.570796, 1.664181],accel_mss,speed_ms,0,blend_radius_m)
    movel([0.093901, -1.466023, -2.501158, -0.745209, 1.570796, 1.664698],accel_mss,speed_ms,0,blend_radius_m)
    movel([0.094816, -1.466465, -2.500788, -0.745136, 1.570796, 1.665612],accel_mss,speed_ms,0,blend_radius_m)
    movel([0.095859, -1.466661, -2.500625, -0.745103, 1.570796, 1.666655],accel_mss,speed_ms,0,blend_radius_m)
    movel([0.097030, -1.466609, -2.500669, -0.745112, 1.570796, 1.667826],accel_mss,speed_ms,0,blend_radius_m)
    movel([0.098335, -1.466306, -2.500921, -0.745162, 1.570796, 1.669131],accel_mss,speed_ms,0,blend_radius_m)
    movel([0.099693, -1.465776, -2.501364, -0.745249, 1.570796, 1.670489],accel_mss,speed_ms,0,blend_radius_m)
    movel([0.101031, -1.465031, -2.501985, -0.745373, 1.570796, 1.671828],accel_mss,speed_ms,0,blend_radius_m)
    movel([0.102349, -1.464074, -2.502781, -0.745534, 1.570796, 1.673146],accel_mss,speed_ms,0,blend_radius_m)
    movel([0.103652, -1.462901, -2.503755, -0.745732, 1.570796, 1.674448],accel_mss,speed_ms,0,blend_radius_m)
    movel([0.105460, -1.460691, -2.505586, -0.746112, 1.570796, 1.676256],accel_mss,speed_ms,0,blend_radius_m)
    movel([0.106567, -1.458339, -2.507526, -0.746525, 1.570796, 1.677363],accel_mss,speed_ms,0,blend_radius_m)
    movel([0.106833, -1.457125, -2.508524, -0.746741, 1.570796, 1.677629],accel_mss,speed_ms,0,blend_radius_m)
    movel([0.106875, -1.455909, -2.509520, -0.746960, 1.570796, 1.677671],accel_mss,speed_ms,0,blend_radius_m)
    movel([0.106293, -1.453467, -2.511516, -0.747406, 1.570796, 1.677089],accel_mss,speed_ms,0,blend_radius_m)
    movel([0.104760, -1.451110, -2.513434, -0.747846, 1.570796, 1.675557],accel_mss,speed_ms,0,blend_radius_m)
    movel([0.102219, -1.448940, -2.515191, -0.748258, 1.570796, 1.673015],accel_mss,speed_ms,0,blend_radius_m)
    movel([0.112879, -1.438335, -2.523679, -0.750375, 1.570796, 1.683675],accel_mss,speed_ms,0,blend_radius_m)
    movel([0.125357, -1.447246, -2.516558, -0.748584, 1.570796, 1.696153],accel_mss,speed_ms,0,blend_radius_m)
    movel([0.118375, -1.454033, -2.511054, -0.747302, 1.570796, 1.689171],accel_mss,speed_ms,0,blend_radius_m)
    movel([0.119565, -1.452078, -2.512647, -0.747664, 1.570796, 1.690361],accel_mss,speed_ms,0,blend_radius_m)
    movel([0.120216, -1.449982, -2.514348, -0.748059, 1.570796, 1.691012],accel_mss,speed_ms,0,blend_radius_m)
    movel([0.120286, -1.447853, -2.516069, -0.748467, 1.570796, 1.691082],accel_mss,speed_ms,0,blend_radius_m)
    movel([0.119744, -1.445795, -2.517726, -0.748868, 1.570796, 1.690540],accel_mss,speed_ms,0,blend_radius_m)
    movel([0.118574, -1.443902, -2.519245, -0.749242, 1.570796, 1.689371],accel_mss,speed_ms,0,blend_radius_m)
    movel([0.116776, -1.442270, -2.520550, -0.749569, 1.570796, 1.687572],accel_mss,speed_ms,0,blend_radius_m)
    movel([0.108891, -1.450046, -2.514296, -0.748047, 1.570796, 1.679687],accel_mss,speed_ms,0,blend_radius_m)
    movel([0.111149, -1.451987, -2.512721, -0.747681, 1.570796, 1.681946],accel_mss,speed_ms,0,blend_radius_m)
    movel([0.112862, -1.454281, -2.510852, -0.747256, 1.570796, 1.683658],accel_mss,speed_ms,0,blend_radius_m)
    movel([0.113843, -1.456836, -2.508760, -0.746793, 1.570796, 1.684640],accel_mss,speed_ms,0,blend_radius_m)
    movel([0.113996, -1.458177, -2.507659, -0.746553, 1.570796, 1.684792],accel_mss,speed_ms,0,blend_radius_m)
    movel([0.113921, -1.459562, -2.506518, -0.746309, 1.570796, 1.684717],accel_mss,speed_ms,0,blend_radius_m)
    movel([0.113584, -1.460961, -2.505363, -0.746065, 1.570796, 1.684380],accel_mss,speed_ms,0,blend_radius_m)
    movel([0.112946, -1.462346, -2.504216, -0.745827, 1.570796, 1.683742],accel_mss,speed_ms,0,blend_radius_m)
    movel([0.112010, -1.463719, -2.503077, -0.745594, 1.570796, 1.682807],accel_mss,speed_ms,0,blend_radius_m)
    movel([0.110776, -1.465079, -2.501945, -0.745365, 1.570796, 1.681573],accel_mss,speed_ms,0,blend_radius_m)
    movel([0.109370, -1.466315, -2.500914, -0.745160, 1.570796, 1.680166],accel_mss,speed_ms,0,blend_radius_m)
    movel([0.107913, -1.467322, -2.500072, -0.744995, 1.570796, 1.678709],accel_mss,speed_ms,0,blend_radius_m)
    movel([0.106405, -1.468100, -2.499420, -0.744868, 1.570796, 1.677201],accel_mss,speed_ms,0,blend_radius_m)
    movel([0.104842, -1.468651, -2.498959, -0.744779, 1.570796, 1.675639],accel_mss,speed_ms,0,blend_radius_m)
    movel([0.101726, -1.469166, -2.498526, -0.744696, 1.570796, 1.672522],accel_mss,speed_ms,0,blend_radius_m)
    movel([0.098732, -1.468965, -2.498695, -0.744729, 1.570796, 1.669529],accel_mss,speed_ms,0,blend_radius_m)
    movel([0.095976, -1.468176, -2.499357, -0.744856, 1.570796, 1.666772],accel_mss,speed_ms,0,blend_radius_m)
    movel([0.093579, -1.466926, -2.500403, -0.745060, 1.570796, 1.664375],accel_mss,speed_ms,0,blend_radius_m)
    movel([0.092215, -1.465786, -2.501355, -0.745248, 1.570796, 1.663012],accel_mss,speed_ms,0,blend_radius_m)
    movel([0.091101, -1.464365, -2.502539, -0.745485, 1.570796, 1.661898],accel_mss,speed_ms,0,blend_radius_m)
    movel([0.090369, -1.462764, -2.503870, -0.745756, 1.570796, 1.661165],accel_mss,speed_ms,0,blend_radius_m)
    movel([0.090161, -1.461082, -2.505263, -0.746044, 1.570796, 1.660957],accel_mss,speed_ms,0,blend_radius_m)
    movel([0.090557, -1.459431, -2.506626, -0.746332, 1.570796, 1.661353],accel_mss,speed_ms,0,blend_radius_m)
    movel([0.091644, -1.457915, -2.507874, -0.746600, 1.570796, 1.662440],accel_mss,speed_ms,0,blend_radius_m)
    speed_ms = 0.003
    movel([0.091644, -1.451861, -2.505107, -0.755421, 1.570796, 1.662440],accel_mss,speed_ms,0,blend_radius_m)
    speed_ms = 0.05
    movel([0.091644, -1.428444, -2.493753, -0.790192, 1.570796, 1.662440],accel_mss,speed_ms,0,blend_radius_m)
    #M_RunCode9
    movel([0.060488, -1.370560, -2.536857, -0.804973, 1.570796, 1.631284],accel_mss,speed_ms,0,blend_radius_m)
    #M_RunCode3
    movel([0.060488, -1.395107, -2.548924, -0.768359, 1.570796, 1.631284],accel_mss,speed_ms,0,blend_radius_m)
    speed_ms = 0.003
    movel([0.060488, -1.401474, -2.551869, -0.759046, 1.570796, 1.631284],accel_mss,speed_ms,0,blend_radius_m)
    speed_ms = 0.02
    movel([0.057912, -1.402882, -2.550829, -0.758678, 1.570796, 1.628708],accel_mss,speed_ms,0,blend_radius_m)
    movel([0.055150, -1.403883, -2.550088, -0.758418, 1.570796, 1.625946],accel_mss,speed_ms,0,blend_radius_m)
    movel([0.052304, -1.404524, -2.549612, -0.758252, 1.570796, 1.623100],accel_mss,speed_ms,0,blend_radius_m)
    movel([0.049478, -1.404845, -2.549374, -0.758170, 1.570796, 1.620274],accel_mss,speed_ms,0,blend_radius_m)
    movel([0.046779, -1.404883, -2.549346, -0.758160, 1.570796, 1.617575],accel_mss,speed_ms,0,blend_radius_m)
    movel([0.046830, -1.402197, -2.551335, -0.758857, 1.570796, 1.617627],accel_mss,speed_ms,0,blend_radius_m)
    movel([0.047701, -1.399025, -2.553670, -0.759694, 1.570796, 1.618497],accel_mss,speed_ms,0,blend_radius_m)
    movel([0.049282, -1.395655, -2.556135, -0.760599, 1.570796, 1.620078],accel_mss,speed_ms,0,blend_radius_m)
    movel([0.051452, -1.392398, -2.558502, -0.761489, 1.570796, 1.622248],accel_mss,speed_ms,0,blend_radius_m)
    movel([0.054094, -1.389561, -2.560551, -0.762277, 1.570796, 1.624891],accel_mss,speed_ms,0,blend_radius_m)
    movel([0.055551, -1.388400, -2.561386, -0.762603, 1.570796, 1.626347],accel_mss,speed_ms,0,blend_radius_m)
    movel([0.057075, -1.387463, -2.562058, -0.762868, 1.570796, 1.627871],accel_mss,speed_ms,0,blend_radius_m)
    movel([0.058652, -1.386791, -2.562540, -0.763058, 1.570796, 1.629448],accel_mss,speed_ms,0,blend_radius_m)
    movel([0.060264, -1.386424, -2.562802, -0.763162, 1.570796, 1.631060],accel_mss,speed_ms,0,blend_radius_m)
    movel([0.061891, -1.386400, -2.562820, -0.763169, 1.570796, 1.632687],accel_mss,speed_ms,0,blend_radius_m)
    movel([0.063514, -1.386763, -2.562560, -0.763066, 1.570796, 1.634311],accel_mss,speed_ms,0,blend_radius_m)
    movel([0.065406, -1.387920, -2.561731, -0.762739, 1.570796, 1.636202],accel_mss,speed_ms,0,blend_radius_m)
    movel([0.066409, -1.389653, -2.560484, -0.762252, 1.570796, 1.637205],accel_mss,speed_ms,0,blend_radius_m)
    movel([0.066594, -1.391847, -2.558900, -0.761641, 1.570796, 1.637391],accel_mss,speed_ms,0,blend_radius_m)
    movel([0.066032, -1.394384, -2.557060, -0.760944, 1.570796, 1.636828],accel_mss,speed_ms,0,blend_radius_m)
    movel([0.064655, -1.397272, -2.554954, -0.760162, 1.570796, 1.635452],accel_mss,speed_ms,0,blend_radius_m)
    movel([0.062771, -1.399619, -2.553234, -0.759536, 1.570796, 1.633568],accel_mss,speed_ms,0,blend_radius_m)
    movel([0.060488, -1.401474, -2.551869, -0.759046, 1.570796, 1.631284],accel_mss,speed_ms,0,blend_radius_m)
    speed_ms = 0.003
    movel([0.060488, -1.395107, -2.548924, -0.768359, 1.570796, 1.631284],accel_mss,speed_ms,0,blend_radius_m)
    speed_ms = 0.05
    movel([0.060488, -1.370560, -2.536857, -0.804973, 1.570796, 1.631284],accel_mss,speed_ms,0,blend_radius_m)
    #M_RunCode9
    movel([0.102810, -1.281657, -2.594206, -0.836526, 1.570796, 1.673607],accel_mss,speed_ms,0,blend_radius_m)
    #M_RunCode3
    movel([0.102810, -1.307703, -2.607417, -0.797270, 1.570796, 1.673607],accel_mss,speed_ms,0,blend_radius_m)
    speed_ms = 0.003
    movel([0.102810, -1.314498, -2.610649, -0.787241, 1.570796, 1.673607],accel_mss,speed_ms,0,blend_radius_m)
    speed_ms = 0.007
    movel([0.101124, -1.314285, -2.610781, -0.787324, 1.570796, 1.671920],accel_mss,speed_ms,0,blend_radius_m)
    movel([0.099693, -1.313627, -2.611185, -0.787576, 1.570796, 1.670490],accel_mss,speed_ms,0,blend_radius_m)
    movel([0.098422, -1.312733, -2.611735, -0.787921, 1.570796, 1.669218],accel_mss,speed_ms,0,blend_radius_m)
    movel([0.099152, -1.312243, -2.612036, -0.788110, 1.570796, 1.669948],accel_mss,speed_ms,0,blend_radius_m)
    movel([0.099808, -1.312246, -2.612034, -0.788109, 1.570796, 1.670605],accel_mss,speed_ms,0,blend_radius_m)
    movel([0.100590, -1.312198, -2.612063, -0.788128, 1.570796, 1.671386],accel_mss,speed_ms,0,blend_radius_m)
    movel([0.101690, -1.311561, -2.612454, -0.788374, 1.570796, 1.672486],accel_mss,speed_ms,0,blend_radius_m)
    movel([0.102667, -1.310546, -2.613075, -0.788768, 1.570796, 1.673464],accel_mss,speed_ms,0,blend_radius_m)
    movel([0.103478, -1.309414, -2.613765, -0.789209, 1.570796, 1.674274],accel_mss,speed_ms,0,blend_radius_m)
    movel([0.104551, -1.307819, -2.614737, -0.789834, 1.570796, 1.675348],accel_mss,speed_ms,0,blend_radius_m)
    movel([0.103059, -1.306582, -2.615487, -0.790320, 1.570796, 1.673855],accel_mss,speed_ms,0,blend_radius_m)
    movel([0.101322, -1.306101, -2.615778, -0.790510, 1.570796, 1.672118],accel_mss,speed_ms,0,blend_radius_m)
    movel([0.100360, -1.306234, -2.615698, -0.790457, 1.570796, 1.671156],accel_mss,speed_ms,0,blend_radius_m)
    movel([0.099335, -1.306666, -2.615436, -0.790287, 1.570796, 1.670132],accel_mss,speed_ms,0,blend_radius_m)
    movel([0.098248, -1.307435, -2.614970, -0.789985, 1.570796, 1.669044],accel_mss,speed_ms,0,blend_radius_m)
    movel([0.097100, -1.308574, -2.614277, -0.789538, 1.570796, 1.667896],accel_mss,speed_ms,0,blend_radius_m)
    movel([0.096912, -1.307374, -2.615007, -0.790008, 1.570796, 1.667709],accel_mss,speed_ms,0,blend_radius_m)
    movel([0.096937, -1.306264, -2.615679, -0.790445, 1.570796, 1.667734],accel_mss,speed_ms,0,blend_radius_m)
    movel([0.097128, -1.305794, -2.615964, -0.790631, 1.570796, 1.667925],accel_mss,speed_ms,0,blend_radius_m)
    movel([0.097494, -1.305410, -2.616196, -0.790783, 1.570796, 1.668290],accel_mss,speed_ms,0,blend_radius_m)
    movel([0.098903, -1.304980, -2.616456, -0.790953, 1.570796, 1.669699],accel_mss,speed_ms,0,blend_radius_m)
    movel([0.101602, -1.305034, -2.616424, -0.790932, 1.570796, 1.672398],accel_mss,speed_ms,0,blend_radius_m)
    movel([0.104000, -1.305726, -2.616005, -0.790658, 1.570796, 1.674796],accel_mss,speed_ms,0,blend_radius_m)
    movel([0.104911, -1.306348, -2.615629, -0.790412, 1.570796, 1.675707],accel_mss,speed_ms,0,blend_radius_m)
    movel([0.105534, -1.307180, -2.615125, -0.790085, 1.570796, 1.676331],accel_mss,speed_ms,0,blend_radius_m)
    movel([0.105803, -1.308230, -2.614487, -0.789673, 1.570796, 1.676600],accel_mss,speed_ms,0,blend_radius_m)
    movel([0.105647, -1.309515, -2.613704, -0.789170, 1.570796, 1.676443],accel_mss,speed_ms,0,blend_radius_m)
    movel([0.103926, -1.309531, -2.613694, -0.789164, 1.570796, 1.674722],accel_mss,speed_ms,0,blend_radius_m)
    movel([0.104851, -1.314057, -2.610921, -0.787411, 1.570796, 1.675647],accel_mss,speed_ms,0,blend_radius_m)
    movel([0.102810, -1.314498, -2.610649, -0.787241, 1.570796, 1.673607],accel_mss,speed_ms,0,blend_radius_m)
    speed_ms = 0.003
    movel([0.102810, -1.307703, -2.607417, -0.797270, 1.570796, 1.673607],accel_mss,speed_ms,0,blend_radius_m)
    speed_ms = 0.05
    movel([0.102810, -1.281657, -2.594206, -0.836526, 1.570796, 1.673607],accel_mss,speed_ms,0,blend_radius_m)
    #M_RunCode9
    movel([0.062673, -1.265901, -2.603322, -0.843166, 1.570796, 1.633469],accel_mss,speed_ms,0,blend_radius_m)
    #M_RunCode3
    movel([0.062673, -1.292173, -2.616738, -0.803478, 1.570796, 1.633469],accel_mss,speed_ms,0,blend_radius_m)
    speed_ms = 0.003
    movel([0.062673, -1.299035, -2.620023, -0.793331, 1.570796, 1.633469],accel_mss,speed_ms,0,blend_radius_m)
    speed_ms = 0.02
    movel([0.060971, -1.301295, -2.618672, -0.792422, 1.570796, 1.631768],accel_mss,speed_ms,0,blend_radius_m)
    movel([0.059037, -1.303474, -2.617364, -0.791551, 1.570796, 1.629833],accel_mss,speed_ms,0,blend_radius_m)
    movel([0.056880, -1.305538, -2.616119, -0.790732, 1.570796, 1.627676],accel_mss,speed_ms,0,blend_radius_m)
    movel([0.054516, -1.307458, -2.614956, -0.789975, 1.570796, 1.625312],accel_mss,speed_ms,0,blend_radius_m)
    movel([0.051966, -1.309202, -2.613895, -0.789292, 1.570796, 1.622762],accel_mss,speed_ms,0,blend_radius_m)
    movel([0.050531, -1.309908, -2.613464, -0.789017, 1.570796, 1.621327],accel_mss,speed_ms,0,blend_radius_m)
    movel([0.048992, -1.310471, -2.613121, -0.788798, 1.570796, 1.619788],accel_mss,speed_ms,0,blend_radius_m)
    movel([0.047608, -1.310986, -2.612806, -0.788597, 1.570796, 1.618404],accel_mss,speed_ms,0,blend_radius_m)
    movel([0.046652, -1.311534, -2.612470, -0.788385, 1.570796, 1.617448],accel_mss,speed_ms,0,blend_radius_m)
    movel([0.045483, -1.312989, -2.611578, -0.787822, 1.570796, 1.616280],accel_mss,speed_ms,0,blend_radius_m)
    movel([0.044130, -1.315113, -2.610270, -0.787006, 1.570796, 1.614926],accel_mss,speed_ms,0,blend_radius_m)
    movel([0.042745, -1.317335, -2.608896, -0.786158, 1.570796, 1.613542],accel_mss,speed_ms,0,blend_radius_m)
    movel([0.041473, -1.319096, -2.607802, -0.785491, 1.570796, 1.612270],accel_mss,speed_ms,0,blend_radius_m)
    movel([0.038551, -1.322121, -2.605913, -0.784355, 1.570796, 1.609348],accel_mss,speed_ms,0,blend_radius_m)
    movel([0.035652, -1.324487, -2.604427, -0.783475, 1.570796, 1.606448],accel_mss,speed_ms,0,blend_radius_m)
    movel([0.032775, -1.326262, -2.603308, -0.782820, 1.570796, 1.603571],accel_mss,speed_ms,0,blend_radius_m)
    movel([0.029921, -1.327506, -2.602520, -0.782363, 1.570796, 1.600718],accel_mss,speed_ms,0,blend_radius_m)
    movel([0.027098, -1.328280, -2.602030, -0.782080, 1.570796, 1.597894],accel_mss,speed_ms,0,blend_radius_m)
    movel([0.024310, -1.328639, -2.601801, -0.781948, 1.570796, 1.595106],accel_mss,speed_ms,0,blend_radius_m)
    movel([0.021561, -1.328641, -2.601800, -0.781948, 1.570796, 1.592357],accel_mss,speed_ms,0,blend_radius_m)
    movel([0.018855, -1.328342, -2.601990, -0.782057, 1.570796, 1.589651],accel_mss,speed_ms,0,blend_radius_m)
    movel([0.013608, -1.327062, -2.602802, -0.782526, 1.570796, 1.584405],accel_mss,speed_ms,0,blend_radius_m)
    movel([0.008640, -1.325228, -2.603960, -0.783201, 1.570796, 1.579436],accel_mss,speed_ms,0,blend_radius_m)
    movel([-0.000140, -1.321616, -2.606229, -0.784544, 1.570796, 1.570657],accel_mss,speed_ms,0,blend_radius_m)
    movel([-0.004320, -1.320469, -2.606946, -0.784974, 1.570796, 1.566476],accel_mss,speed_ms,0,blend_radius_m)
    movel([-0.009452, -1.319595, -2.607491, -0.785303, 1.570796, 1.561344],accel_mss,speed_ms,0,blend_radius_m)
    movel([-0.015283, -1.319073, -2.607816, -0.785500, 1.570796, 1.555514],accel_mss,speed_ms,0,blend_radius_m)
    movel([-0.021548, -1.318977, -2.607875, -0.785536, 1.570796, 1.549248],accel_mss,speed_ms,0,blend_radius_m)
    movel([-0.027979, -1.319376, -2.607627, -0.785386, 1.570796, 1.542817],accel_mss,speed_ms,0,blend_radius_m)
    movel([-0.034301, -1.320323, -2.607037, -0.785029, 1.570796, 1.536495],accel_mss,speed_ms,0,blend_radius_m)
    movel([-0.040235, -1.321867, -2.606072, -0.784450, 1.570796, 1.530561],accel_mss,speed_ms,0,blend_radius_m)
    movel([-0.042969, -1.322877, -2.605439, -0.784073, 1.570796, 1.527828],accel_mss,speed_ms,0,blend_radius_m)
    movel([-0.045502, -1.324050, -2.604702, -0.783637, 1.570796, 1.525295],accel_mss,speed_ms,0,blend_radius_m)
    movel([-0.048048, -1.325495, -2.603792, -0.783102, 1.570796, 1.522749],accel_mss,speed_ms,0,blend_radius_m)
    movel([-0.050940, -1.327387, -2.602596, -0.782406, 1.570796, 1.519856],accel_mss,speed_ms,0,blend_radius_m)
    movel([-0.053974, -1.329660, -2.601152, -0.781576, 1.570796, 1.516823],accel_mss,speed_ms,0,blend_radius_m)
    movel([-0.056949, -1.332244, -2.599503, -0.780642, 1.570796, 1.513848],accel_mss,speed_ms,0,blend_radius_m)
    movel([-0.059657, -1.335061, -2.597695, -0.779633, 1.570796, 1.511139],accel_mss,speed_ms,0,blend_radius_m)
    movel([-0.061909, -1.338046, -2.595768, -0.778576, 1.570796, 1.508888],accel_mss,speed_ms,0,blend_radius_m)
    movel([-0.063504, -1.341126, -2.593765, -0.777497, 1.570796, 1.507292],accel_mss,speed_ms,0,blend_radius_m)
    movel([-0.063999, -1.342680, -2.592751, -0.776958, 1.570796, 1.506798],accel_mss,speed_ms,0,blend_radius_m)
    movel([-0.064257, -1.344233, -2.591733, -0.776423, 1.570796, 1.506539],accel_mss,speed_ms,0,blend_radius_m)
    movel([-0.064091, -1.346436, -2.590284, -0.775669, 1.570796, 1.506706],accel_mss,speed_ms,0,blend_radius_m)
    movel([-0.063209, -1.348011, -2.589244, -0.775134, 1.570796, 1.507587],accel_mss,speed_ms,0,blend_radius_m)
    movel([-0.061697, -1.349027, -2.588571, -0.774791, 1.570796, 1.509100],accel_mss,speed_ms,0,blend_radius_m)
    movel([-0.059635, -1.349546, -2.588227, -0.774616, 1.570796, 1.511162],accel_mss,speed_ms,0,blend_radius_m)
    movel([-0.057103, -1.349631, -2.588170, -0.774588, 1.570796, 1.513693],accel_mss,speed_ms,0,blend_radius_m)
    movel([-0.054182, -1.349345, -2.588360, -0.774684, 1.570796, 1.516614],accel_mss,speed_ms,0,blend_radius_m)
    movel([-0.050947, -1.348746, -2.588757, -0.774886, 1.570796, 1.519849],accel_mss,speed_ms,0,blend_radius_m)
    movel([-0.047477, -1.347898, -2.589319, -0.775172, 1.570796, 1.523319],accel_mss,speed_ms,0,blend_radius_m)
    movel([-0.040154, -1.345684, -2.590779, -0.775926, 1.570796, 1.530642],accel_mss,speed_ms,0,blend_radius_m)
    movel([-0.032847, -1.343171, -2.592429, -0.776789, 1.570796, 1.537949],accel_mss,speed_ms,0,blend_radius_m)
    movel([-0.026213, -1.340819, -2.593966, -0.777605, 1.570796, 1.544584],accel_mss,speed_ms,0,blend_radius_m)
    movel([-0.020917, -1.339093, -2.595088, -0.778208, 1.570796, 1.549880],accel_mss,speed_ms,0,blend_radius_m)
    movel([-0.008098, -1.335388, -2.597485, -0.779517, 1.570796, 1.562698],accel_mss,speed_ms,0,blend_radius_m)
    movel([-0.001242, -1.333585, -2.598644, -0.780160, 1.570796, 1.569554],accel_mss,speed_ms,0,blend_radius_m)
    movel([0.004075, -1.332484, -2.599350, -0.780556, 1.570796, 1.574872],accel_mss,speed_ms,0,blend_radius_m)
    movel([0.006089, -1.332313, -2.599459, -0.780617, 1.570796, 1.576885],accel_mss,speed_ms,0,blend_radius_m)
    movel([0.007962, -1.332384, -2.599414, -0.780592, 1.570796, 1.578758],accel_mss,speed_ms,0,blend_radius_m)
    movel([0.011274, -1.333194, -2.598895, -0.780300, 1.570796, 1.582071],accel_mss,speed_ms,0,blend_radius_m)
    movel([0.014005, -1.334783, -2.597874, -0.779732, 1.570796, 1.584801],accel_mss,speed_ms,0,blend_radius_m)
    movel([0.016157, -1.337009, -2.596439, -0.778942, 1.570796, 1.586953],accel_mss,speed_ms,0,blend_radius_m)
    movel([0.017725, -1.339735, -2.594671, -0.777983, 1.570796, 1.588521],accel_mss,speed_ms,0,blend_radius_m)
    movel([0.018714, -1.342828, -2.592654, -0.776907, 1.570796, 1.589510],accel_mss,speed_ms,0,blend_radius_m)
    movel([0.019132, -1.346151, -2.590472, -0.775766, 1.570796, 1.589928],accel_mss,speed_ms,0,blend_radius_m)
    movel([0.018983, -1.349568, -2.588212, -0.774609, 1.570796, 1.589779],accel_mss,speed_ms,0,blend_radius_m)
    movel([0.018040, -1.353888, -2.585332, -0.773169, 1.570796, 1.588836],accel_mss,speed_ms,0,blend_radius_m)
    movel([0.017330, -1.355729, -2.584097, -0.772563, 1.570796, 1.588126],accel_mss,speed_ms,0,blend_radius_m)
    movel([0.016466, -1.357392, -2.582978, -0.772019, 1.570796, 1.587262],accel_mss,speed_ms,0,blend_radius_m)
    movel([0.015462, -1.358898, -2.581961, -0.771531, 1.570796, 1.586259],accel_mss,speed_ms,0,blend_radius_m)
    movel([0.014321, -1.360271, -2.581030, -0.771088, 1.570796, 1.585118],accel_mss,speed_ms,0,blend_radius_m)
    movel([0.011664, -1.362722, -2.579363, -0.770304, 1.570796, 1.582460],accel_mss,speed_ms,0,blend_radius_m)
    movel([0.008551, -1.364931, -2.577853, -0.769605, 1.570796, 1.579347],accel_mss,speed_ms,0,blend_radius_m)
    movel([0.005045, -1.367086, -2.576374, -0.768929, 1.570796, 1.575842],accel_mss,speed_ms,0,blend_radius_m)
    movel([-0.002899, -1.371950, -2.573010, -0.767429, 1.570796, 1.567897],accel_mss,speed_ms,0,blend_radius_m)
    movel([-0.003291, -1.372227, -2.572817, -0.767344, 1.570796, 1.567506],accel_mss,speed_ms,0,blend_radius_m)
    movel([-0.003098, -1.372226, -2.572818, -0.767345, 1.570796, 1.567698],accel_mss,speed_ms,0,blend_radius_m)
    movel([-0.001268, -1.371533, -2.573300, -0.767556, 1.570796, 1.569529],accel_mss,speed_ms,0,blend_radius_m)
    movel([0.006076, -1.368405, -2.575465, -0.768519, 1.570796, 1.576872],accel_mss,speed_ms,0,blend_radius_m)
    movel([0.018333, -1.363222, -2.579022, -0.770145, 1.570796, 1.589129],accel_mss,speed_ms,0,blend_radius_m)
    movel([0.012601, -1.368195, -2.575610, -0.768584, 1.570796, 1.583397],accel_mss,speed_ms,0,blend_radius_m)
    movel([0.006067, -1.373477, -2.571947, -0.766964, 1.570796, 1.576863],accel_mss,speed_ms,0,blend_radius_m)
    movel([-0.000996, -1.378907, -2.568141, -0.765341, 1.570796, 1.569801],accel_mss,speed_ms,0,blend_radius_m)
    movel([-0.008330, -1.384316, -2.564308, -0.763765, 1.570796, 1.562466],accel_mss,speed_ms,0,blend_radius_m)
    movel([-0.022815, -1.394452, -2.557011, -0.760926, 1.570796, 1.547982],accel_mss,speed_ms,0,blend_radius_m)
    movel([-0.029489, -1.398858, -2.553793, -0.759738, 1.570796, 1.541307],accel_mss,speed_ms,0,blend_radius_m)
    movel([-0.035482, -1.402621, -2.551022, -0.758746, 1.570796, 1.535314],accel_mss,speed_ms,0,blend_radius_m)
    movel([-0.042163, -1.410108, -2.545446, -0.756834, 1.570796, 1.528633],accel_mss,speed_ms,0,blend_radius_m)
    movel([-0.048670, -1.417962, -2.539510, -0.754918, 1.570796, 1.522126],accel_mss,speed_ms,0,blend_radius_m)
    movel([-0.061315, -1.434043, -2.527066, -0.751280, 1.570796, 1.509481],accel_mss,speed_ms,0,blend_radius_m)
    movel([-0.067546, -1.441940, -2.520813, -0.749636, 1.570796, 1.503251],accel_mss,speed_ms,0,blend_radius_m)
    movel([-0.073784, -1.449537, -2.514708, -0.748144, 1.570796, 1.497012],accel_mss,speed_ms,0,blend_radius_m)
    movel([-0.080081, -1.456689, -2.508881, -0.746819, 1.570796, 1.490715],accel_mss,speed_ms,0,blend_radius_m)
    movel([-0.086500, -1.463258, -2.503460, -0.745672, 1.570796, 1.484296],accel_mss,speed_ms,0,blend_radius_m)
    movel([-0.089113, -1.465618, -2.501495, -0.745276, 1.570796, 1.481683],accel_mss,speed_ms,0,blend_radius_m)
    movel([-0.091712, -1.467683, -2.499770, -0.744936, 1.570796, 1.479084],accel_mss,speed_ms,0,blend_radius_m)
    movel([-0.094276, -1.469447, -2.498291, -0.744651, 1.570796, 1.476521],accel_mss,speed_ms,0,blend_radius_m)
    movel([-0.096785, -1.470911, -2.497060, -0.744419, 1.570796, 1.474011],accel_mss,speed_ms,0,blend_radius_m)
    movel([-0.099225, -1.472066, -2.496085, -0.744237, 1.570796, 1.471572],accel_mss,speed_ms,0,blend_radius_m)
    movel([-0.101576, -1.472911, -2.495372, -0.744106, 1.570796, 1.469221],accel_mss,speed_ms,0,blend_radius_m)
    movel([-0.103820, -1.473442, -2.494923, -0.744024, 1.570796, 1.466976],accel_mss,speed_ms,0,blend_radius_m)
    movel([-0.105937, -1.473654, -2.494744, -0.743992, 1.570796, 1.464859],accel_mss,speed_ms,0,blend_radius_m)
    movel([-0.107910, -1.473539, -2.494841, -0.744009, 1.570796, 1.462887],accel_mss,speed_ms,0,blend_radius_m)
    movel([-0.109720, -1.473091, -2.495220, -0.744078, 1.570796, 1.461076],accel_mss,speed_ms,0,blend_radius_m)
    movel([-0.111344, -1.472304, -2.495885, -0.744200, 1.570796, 1.459452],accel_mss,speed_ms,0,blend_radius_m)
    movel([-0.112768, -1.471173, -2.496839, -0.744377, 1.570796, 1.458028],accel_mss,speed_ms,0,blend_radius_m)
    movel([-0.113968, -1.469686, -2.498090, -0.744613, 1.570796, 1.456829],accel_mss,speed_ms,0,blend_radius_m)
    movel([-0.114922, -1.467834, -2.499643, -0.744912, 1.570796, 1.455875],accel_mss,speed_ms,0,blend_radius_m)
    movel([-0.115609, -1.465610, -2.501502, -0.745277, 1.570796, 1.455187],accel_mss,speed_ms,0,blend_radius_m)
    movel([-0.116006, -1.463000, -2.503674, -0.745715, 1.570796, 1.454790],accel_mss,speed_ms,0,blend_radius_m)
    movel([-0.112936, -1.462764, -2.503869, -0.745756, 1.570796, 1.457860],accel_mss,speed_ms,0,blend_radius_m)
    movel([-0.111418, -1.462572, -2.504029, -0.745788, 1.570796, 1.459378],accel_mss,speed_ms,0,blend_radius_m)
    movel([-0.109924, -1.462088, -2.504430, -0.745871, 1.570796, 1.460872],accel_mss,speed_ms,0,blend_radius_m)
    movel([-0.108807, -1.461396, -2.505003, -0.745990, 1.570796, 1.461989],accel_mss,speed_ms,0,blend_radius_m)
    movel([-0.107556, -1.460330, -2.505884, -0.746175, 1.570796, 1.463241],accel_mss,speed_ms,0,blend_radius_m)
    movel([-0.104733, -1.457261, -2.508412, -0.746717, 1.570796, 1.466063],accel_mss,speed_ms,0,blend_radius_m)
